// TIA Portal V19 export
FUNCTION_BLOCK "HMI_A04_FB"   // FB117, LAD
TITLE = HMI Managment
AUTHOR : Piemme
FAMILY : System
// stored: MemoryReserve 100, SetENOAutomatically false
   VAR_OUTPUT
      MB4_LpJog : Bool;
   END_VAR
   VAR
      MB4_Decoder { ExternalAccessible := 'False'; ExternalVisible := 'False'; ExternalWritable := 'False'} : "ButtonsHMIDecoder";
   END_VAR
   VAR CONSTANT
      "3002_TRASPORTO" : Int := 3002;
      "3011_FERMI_P1" : Int := 3011;
      "3012_FERMI_P1_SFALSATORE" : Int := 3012;
      "3021_FERMI_P2" : Int := 3021;
      "3022_FERMI_P2_SOLLEVATORE" : Int := 3022;
      "3031_FERMI_P3" : Int := 3031;
      "3032_SOLLEVA_RIBALTA" : Int := 3032;
      "3033_ROT_RIBALTA" : Int := 3033;
      "3041_FERMI_P4" : Int := 3041;
      "3042_SPINTORE_LAT_VRT_P5" : Int := 3042;
      "3043_SPINTORE_LAT_ORZ_P5" : Int := 3043;
      "3044_SOLLEVATORI_P5" : Int := 3044;
      "3045_SPINTORE_LAT_OP" : Int := 3045;
      "3051_RIBALTATORE_OP-POS0" : Int := 3051;
      "3052_RIBALTATORE_OP-POS1" : Int := 3052;
      "3053_RIBALTATORE_OP-POS2" : Int := 3053;
      "3054_RIBALTATORE_OP-POS3" : Int := 3054;
      "4001_HU_CYTROPACK" : Int := 4001;
      "4011_SPINTORE_OP" : Int := 4011;
      "4012_SPINTORE_AX" : Int := 4012;
      "4013_SPINTORE_VRT" : Int := 4013;
      "4014_SPINTORE_ORZ" : Int := 4014;
      "4021_BORDATRICE_AX" : Int := 4021;
      "4031_RULLIERA_OP" : Int := 4031;
      "4032_RULLIERA_AX" : Int := 4032;
      "4033_BORDATRICE_REG-CASSETTA" : Int := 4033;
      "4034_BORDATRICE_PASS01" : Int := 4034;
      "4035_BORDATRICE_PASS02" : Int := 4035;
      "4036_BORDATRICE_PASS03" : Int := 4036;
      "4037_BORDATRICE_PASS04" : Int := 4037;
      "4038_BORDATRICE_REG-CASSETTA_AX-POS" : Int := 4038;
      "4041_CENTRATORI_OP" : Int := 4041;
      "4042_CENTRATORI_CENTRAGGIO" : Int := 4042;
      "4043_CENTRATORI_SOLLEVAMENTO" : Int := 4043;
      "4051_PAREGGIATORE_CODA_OP" : Int := 4051;
      "4052_PAREGGIATORE_CODA_AX" : Int := 4052;
      "4053_PAREGGIATORE_CODA_BLOCCAGGIO" : Int := 4053;
      "4054_PAREGGIATORE_CODA_BATTUTAVERTICALE" : Int := 4054;
      "4055_PAREGGIATORE_CODA_PAREGGIATORELONGIT" : Int := 4055;
      "4061_PAREGGIATORE_TESTA_OP" : Int := 4061;
      "4062_PAREGGIATORE_TESTA_AX" : Int := 4062;
      "4063_PAREGGIATORE_TESTA_BLOCCAGGIO" : Int := 4063;
      "4064_PAREGGIATORE_TESTA_SOLLEVAMENTO" : Int := 4064;
      "4065_PAREGGIATORE_TESTA_CENTRAGGIO" : Int := 4065;
      "4066_PAREGG_TESTA_AX_POS" : Int := 4066;
      "4067_PAREGG_TESTA_AX_POS" : Int := 4067;
      "4071_MANIPOLATORE_AX" : Int := 4071;
      "4072_MANIPOLATORE_AX-POS" : Int := 4072;
      "4073_MANIPOLATORE_MAGNETE" : Int := 4073;
      "4074_MANIPOLATORE_SOLLEVATORE" : Int := 4074;
      "4080_BORDATRICE_PASS01_LATO-OP" : Int := 4080;
      "4081_BORDATRICE_PASS01_LATO-MOT" : Int := 4081;
      "4082_BORDATRICE_PASS02_LATO-OP" : Int := 4082;
      "4083_BORDATRICE_PASS02_LATO-MOT" : Int := 4083;
      "4084_BORDATRICE_PASS03_LATO-OP" : Int := 4084;
      "4085_BORDATRICE_PASS03_LATO-MOT" : Int := 4085;
      "4086_BORDATRICE_PASS04_LATO-OP" : Int := 4086;
      "4087_BORDATRICE_PASS04_LATO-MOT" : Int := 4087;
      "4088_BORDATRICE_PASS01-COMBO_AX-POS" : Int := 4088;
      "4089_BORDATRICE_PASS02-COMBO_AX-POS" : Int := 4089;
      "4090_BORDATRICE_PASS03-COMBO_AX-POS" : Int := 4090;
      "4091_BORDATRICE_PASS04-COMBO_AX-POS" : Int := 4091;
      "4092_BORDATRICE_PASS01-LATO-OP_AX-POS" : Int := 4092;
      "4093_BORDATRICE_PASS01-LATO-MOT_AX-POS" : Int := 4093;
      "4094_BORDATRICE_PASS02-LATO-OP_AX-POS" : Int := 4094;
      "4095_BORDATRICE_PASS02-LATO-MOT_AX-POS" : Int := 4095;
      "4096_BORDATRICE_PASS03-LATO-OP_AX-POS" : Int := 4096;
      "4097_BORDATRICE_PASS03-LATO-MOT_AX-POS" : Int := 4097;
      "4098_BORDATRICE_PASS04-LATO-OP_AX-POS" : Int := 4098;
      "4099_BORDATRICE_PASS04-LATO-MOT_AX-POS" : Int := 4099;
      "5001_SPALLA_OP_POS" : Int := 5001;
      "5002_SPALLA_TESTA_AX_JOG" : Int := 5002;
      "5003_SPALLA_TESTA_AX_POS" : Int := 5003;
      "5005_SPALLA_CODA_AX" : Int := 5005;
      "5006_SPALLA_CODA_AX_POS" : Int := 5006;
      "5011_SPINTORE_OP" : Int := 5011;
      "5012_SPINTORE_VRT" : Int := 5012;
      "5013_SPINTORE_ORZ" : Int := 5013;
      "5021_TRASLAZIONE_OP_VAI_A_PRELIEVO" : Int := 5021;
      "5022_TRASLAZIONE_OP_PRELIEVO" : Int := 5022;
      "5023_TRASLAZIONE_OP_VAI_A_DEPOSITO" : Int := 5023;
      "5024_TRASLAZIONE_OP_DEPOSITO" : Int := 5024;
      "5025_TRASLAZIONE_AX_JOG" : Int := 5025;
      "5026_TRASLAZIONE_AX_POS" : Int := 5026;
      "5027_TRASLAZIONE_MANIP_SOSTEGNO" : Int := 5027;
      "5028_TRASLAZIONE_MANIP_PAREGGIATORE" : Int := 5028;
      "5029_TRASLAZIONE_SOSTEGNO_VERTICALE" : Int := 5029;
      "5031_SOLLEVAMENTO_OP" : Int := 5031;
      "5032_SOLLEVAMENTO_AX_JOG" : Int := 5032;
      "5033_SOLLEVAMENTO_AX_POS" : Int := 5033;
      "5041_PALETTIANTIRIBALTAMENTO_OP" : Int := 5041;
      "5042_PALETTIANTIRIBALTAMENTO_TESTA_POS0" : Int := 5042;
      "5043_PALETTIANTIRIBALTAMENTO_TESTA_POS1" : Int := 5043;
      "5044_PALETTIANTIRIBALTAMENTO_TESTA_POS2" : Int := 5044;
      "5046_PALETTIANTIRIBALTAMENTO_CODA_POS0" : Int := 5046;
      "5047_PALETTIANTIRIBALTAMENTO_CODA_POS1" : Int := 5047;
      "5048_PALETTIANTIRIBALTAMENTO_CODA_POS2" : Int := 5048;
      "5051_SOSTEGNO_TESTA_AX_JOG" : Int := 5051;
      "5052_SOSTEGNO_TESTA_AX_POS" : Int := 5052;
      "5053_SOSTEGNO_CODA_AX_JOG" : Int := 5053;
      "5054_SOSTEGNO_CODA_AX_POS" : Int := 5054;
      "6001_NAVETTA_OP_VAI_A_PRELIEVO" : Int := 6001;
      "6002_NAVETTA_OP_PRELIEVO" : Int := 6002;
      "6003_NAVETTA_OP_VAI_A_DEPOSITO" : Int := 6003;
      "6004_NAVETTA_OP_DEPOSITO" : Int := 6004;
      "6005_NAVETTA_AX" : Int := 6005;
      "6006_NAVETTA_PALETTI_INTERNI" : Int := 6006;
      "6007_NAVETTA_PALETTI_ESTERNI" : Int := 6007;
      "6008_NAVETTA_AX_POS" : Int := 6008;
   END_VAR
   VAR_TEMP   // added for the SCL form of the ladder/FBD networks
      _w1 : Bool;
   END_VAR
BEGIN

REGION Network 2: <<< MB3 MANUALS OPERATIONS >>>
END_REGION

REGION Network 3 (SCL): Reset Op
   #MB4_Decoder.OpEnabled := FALSE;
   #MB4_Decoder.OpRunning := FALSE;
   #MB4_Decoder.OpDone := FALSE;
END_REGION

REGION Network 4: <<<<<<<<< A0303 STAZIONE 3 >>>>>>>>>>>>>
END_REGION

REGION Network 5: MB3 Code 5001- SPALLE - OP
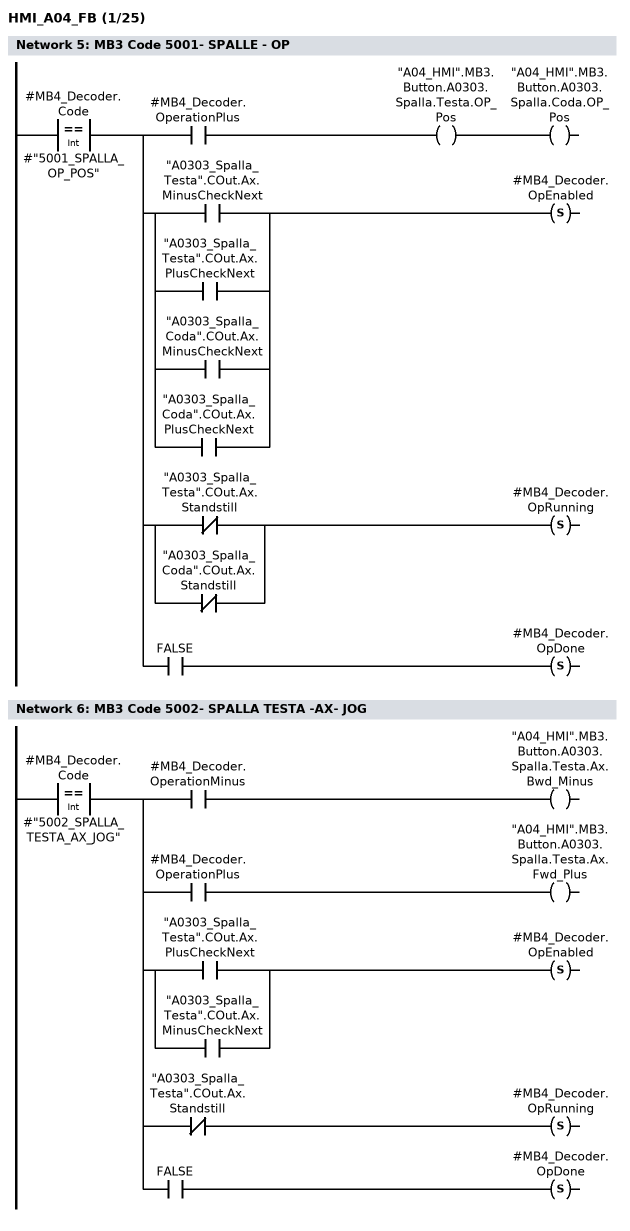
   RUNG wire#powerrail
      { S7_Templates := "SrcType := Int" } EQ_Contact(in1 := #MB4_Decoder.Code, in2 := #"5001_SPALLA_OP_POS")
      wire#w1
      Contact( #MB4_Decoder.OperationPlus )
      Coil( "A04_HMI".MB3.Button.A0303.Spalla.Testa.OP_Pos )
      Coil( "A04_HMI".MB3.Button.A0303.Spalla.Coda.OP_Pos )
   END_RUNG
   RUNG wire#w1
      Contact( "A0303_Spalla_Testa".COut.Ax.MinusCheckNext )
      wire#w2
      S_Coil( #MB4_Decoder.OpEnabled )
   END_RUNG
   RUNG wire#w1
      Contact( "A0303_Spalla_Testa".COut.Ax.PlusCheckNext )
   END_RUNG wire#w2
   RUNG wire#w1
      Contact( "A0303_Spalla_Coda".COut.Ax.MinusCheckNext )
   END_RUNG wire#w2
   RUNG wire#w1
      Contact( "A0303_Spalla_Coda".COut.Ax.PlusCheckNext )
   END_RUNG wire#w2
   RUNG wire#w1
      I_Contact( "A0303_Spalla_Testa".COut.Ax.Standstill )
      wire#w3
      S_Coil( #MB4_Decoder.OpRunning )
   END_RUNG
   RUNG wire#w1
      I_Contact( "A0303_Spalla_Coda".COut.Ax.Standstill )
   END_RUNG wire#w3
   RUNG wire#w1
      Contact( FALSE )
      S_Coil( #MB4_Decoder.OpDone )
   END_RUNG
   // the same network as SCL:
   #_w1 := #MB4_Decoder.Code = #"5001_SPALLA_OP_POS";
   "A04_HMI".MB3.Button.A0303.Spalla.Testa.OP_Pos := #_w1 AND #MB4_Decoder.OperationPlus;
   "A04_HMI".MB3.Button.A0303.Spalla.Coda.OP_Pos := "A04_HMI".MB3.Button.A0303.Spalla.Testa.OP_Pos;
   IF #_w1 AND ("A0303_Spalla_Testa".COut.Ax.MinusCheckNext OR "A0303_Spalla_Testa".COut.Ax.PlusCheckNext OR "A0303_Spalla_Coda".COut.Ax.MinusCheckNext OR "A0303_Spalla_Coda".COut.Ax.PlusCheckNext) THEN
       #MB4_Decoder.OpEnabled := TRUE;
   END_IF;
   IF #_w1 AND (NOT "A0303_Spalla_Testa".COut.Ax.Standstill OR NOT "A0303_Spalla_Coda".COut.Ax.Standstill) THEN
       #MB4_Decoder.OpRunning := TRUE;
   END_IF;
   IF #_w1 AND FALSE THEN #MB4_Decoder.OpDone := TRUE; END_IF;
END_REGION

REGION Network 6: MB3 Code 5002- SPALLA TESTA -AX- JOG
   RUNG wire#powerrail
      { S7_Templates := "SrcType := Int" } EQ_Contact(in1 := #MB4_Decoder.Code, in2 := #"5002_SPALLA_TESTA_AX_JOG")
      wire#w1
      Contact( #MB4_Decoder.OperationMinus )
      Coil( "A04_HMI".MB3.Button.A0303.Spalla.Testa.Ax.Bwd_Minus )
   END_RUNG
   RUNG wire#w1
      Contact( #MB4_Decoder.OperationPlus )
      Coil( "A04_HMI".MB3.Button.A0303.Spalla.Testa.Ax.Fwd_Plus )
   END_RUNG
   RUNG wire#w1
      Contact( "A0303_Spalla_Testa".COut.Ax.PlusCheckNext )
      wire#w2
      S_Coil( #MB4_Decoder.OpEnabled )
   END_RUNG
   RUNG wire#w1
      Contact( "A0303_Spalla_Testa".COut.Ax.MinusCheckNext )
   END_RUNG wire#w2
   RUNG wire#w1
      I_Contact( "A0303_Spalla_Testa".COut.Ax.Standstill )
      S_Coil( #MB4_Decoder.OpRunning )
   END_RUNG
   RUNG wire#w1
      Contact( FALSE )
      S_Coil( #MB4_Decoder.OpDone )
   END_RUNG
   // the same network as SCL:
   #_w1 := #MB4_Decoder.Code = #"5002_SPALLA_TESTA_AX_JOG";
   "A04_HMI".MB3.Button.A0303.Spalla.Testa.Ax.Bwd_Minus := #_w1 AND #MB4_Decoder.OperationMinus;
   "A04_HMI".MB3.Button.A0303.Spalla.Testa.Ax.Fwd_Plus := #_w1 AND #MB4_Decoder.OperationPlus;
   IF #_w1 AND ("A0303_Spalla_Testa".COut.Ax.PlusCheckNext OR "A0303_Spalla_Testa".COut.Ax.MinusCheckNext) THEN
       #MB4_Decoder.OpEnabled := TRUE;
   END_IF;
   IF #_w1 AND NOT "A0303_Spalla_Testa".COut.Ax.Standstill THEN #MB4_Decoder.OpRunning := TRUE; END_IF;
   IF #_w1 AND FALSE THEN #MB4_Decoder.OpDone := TRUE; END_IF;
END_REGION

REGION Network 7: MB3 Code 5003- SPALLA TESTA -AX - POS
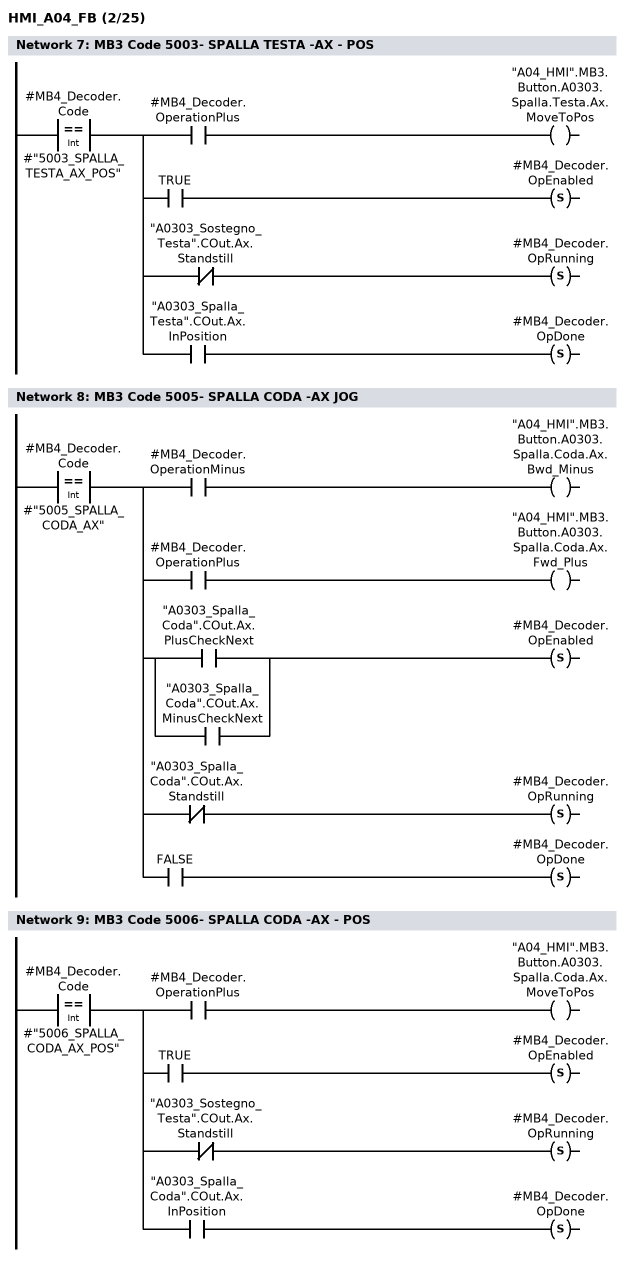
   RUNG wire#powerrail
      { S7_Templates := "SrcType := Int" } EQ_Contact(in1 := #MB4_Decoder.Code, in2 := #"5003_SPALLA_TESTA_AX_POS")
      wire#w1
      Contact( #MB4_Decoder.OperationPlus )
      Coil( "A04_HMI".MB3.Button.A0303.Spalla.Testa.Ax.MoveToPos )
   END_RUNG
   RUNG wire#w1
      Contact( TRUE )
      S_Coil( #MB4_Decoder.OpEnabled )
   END_RUNG
   RUNG wire#w1
      I_Contact( "A0303_Sostegno_Testa".COut.Ax.Standstill )
      S_Coil( #MB4_Decoder.OpRunning )
   END_RUNG
   RUNG wire#w1
      Contact( "A0303_Spalla_Testa".COut.Ax.InPosition )
      S_Coil( #MB4_Decoder.OpDone )
   END_RUNG
   // the same network as SCL:
   #_w1 := #MB4_Decoder.Code = #"5003_SPALLA_TESTA_AX_POS";
   "A04_HMI".MB3.Button.A0303.Spalla.Testa.Ax.MoveToPos := #_w1 AND #MB4_Decoder.OperationPlus;
   IF #_w1 AND TRUE THEN #MB4_Decoder.OpEnabled := TRUE; END_IF;
   IF #_w1 AND NOT "A0303_Sostegno_Testa".COut.Ax.Standstill THEN #MB4_Decoder.OpRunning := TRUE; END_IF;
   IF #_w1 AND "A0303_Spalla_Testa".COut.Ax.InPosition THEN #MB4_Decoder.OpDone := TRUE; END_IF;
END_REGION

REGION Network 8: MB3 Code 5005- SPALLA CODA -AX JOG
   RUNG wire#powerrail
      { S7_Templates := "SrcType := Int" } EQ_Contact(in1 := #MB4_Decoder.Code, in2 := #"5005_SPALLA_CODA_AX")
      wire#w1
      Contact( #MB4_Decoder.OperationMinus )
      Coil( "A04_HMI".MB3.Button.A0303.Spalla.Coda.Ax.Bwd_Minus )
   END_RUNG
   RUNG wire#w1
      Contact( #MB4_Decoder.OperationPlus )
      Coil( "A04_HMI".MB3.Button.A0303.Spalla.Coda.Ax.Fwd_Plus )
   END_RUNG
   RUNG wire#w1
      Contact( "A0303_Spalla_Coda".COut.Ax.PlusCheckNext )
      wire#w2
      S_Coil( #MB4_Decoder.OpEnabled )
   END_RUNG
   RUNG wire#w1
      Contact( "A0303_Spalla_Coda".COut.Ax.MinusCheckNext )
   END_RUNG wire#w2
   RUNG wire#w1
      I_Contact( "A0303_Spalla_Coda".COut.Ax.Standstill )
      S_Coil( #MB4_Decoder.OpRunning )
   END_RUNG
   RUNG wire#w1
      Contact( FALSE )
      S_Coil( #MB4_Decoder.OpDone )
   END_RUNG
   // the same network as SCL:
   #_w1 := #MB4_Decoder.Code = #"5005_SPALLA_CODA_AX";
   "A04_HMI".MB3.Button.A0303.Spalla.Coda.Ax.Bwd_Minus := #_w1 AND #MB4_Decoder.OperationMinus;
   "A04_HMI".MB3.Button.A0303.Spalla.Coda.Ax.Fwd_Plus := #_w1 AND #MB4_Decoder.OperationPlus;
   IF #_w1 AND ("A0303_Spalla_Coda".COut.Ax.PlusCheckNext OR "A0303_Spalla_Coda".COut.Ax.MinusCheckNext) THEN
       #MB4_Decoder.OpEnabled := TRUE;
   END_IF;
   IF #_w1 AND NOT "A0303_Spalla_Coda".COut.Ax.Standstill THEN #MB4_Decoder.OpRunning := TRUE; END_IF;
   IF #_w1 AND FALSE THEN #MB4_Decoder.OpDone := TRUE; END_IF;
END_REGION

REGION Network 9: MB3 Code 5006- SPALLA CODA -AX - POS
   RUNG wire#powerrail
      { S7_Templates := "SrcType := Int" } EQ_Contact(in1 := #MB4_Decoder.Code, in2 := #"5006_SPALLA_CODA_AX_POS")
      wire#w1
      Contact( #MB4_Decoder.OperationPlus )
      Coil( "A04_HMI".MB3.Button.A0303.Spalla.Coda.Ax.MoveToPos )
   END_RUNG
   RUNG wire#w1
      Contact( TRUE )
      S_Coil( #MB4_Decoder.OpEnabled )
   END_RUNG
   RUNG wire#w1
      I_Contact( "A0303_Sostegno_Testa".COut.Ax.Standstill )
      S_Coil( #MB4_Decoder.OpRunning )
   END_RUNG
   RUNG wire#w1
      Contact( "A0303_Spalla_Coda".COut.Ax.InPosition )
      S_Coil( #MB4_Decoder.OpDone )
   END_RUNG
   // the same network as SCL:
   #_w1 := #MB4_Decoder.Code = #"5006_SPALLA_CODA_AX_POS";
   "A04_HMI".MB3.Button.A0303.Spalla.Coda.Ax.MoveToPos := #_w1 AND #MB4_Decoder.OperationPlus;
   IF #_w1 AND TRUE THEN #MB4_Decoder.OpEnabled := TRUE; END_IF;
   IF #_w1 AND NOT "A0303_Sostegno_Testa".COut.Ax.Standstill THEN #MB4_Decoder.OpRunning := TRUE; END_IF;
   IF #_w1 AND "A0303_Spalla_Coda".COut.Ax.InPosition THEN #MB4_Decoder.OpDone := TRUE; END_IF;
END_REGION

REGION Network 10: MB3 Code 5011- SPINTORE- OP
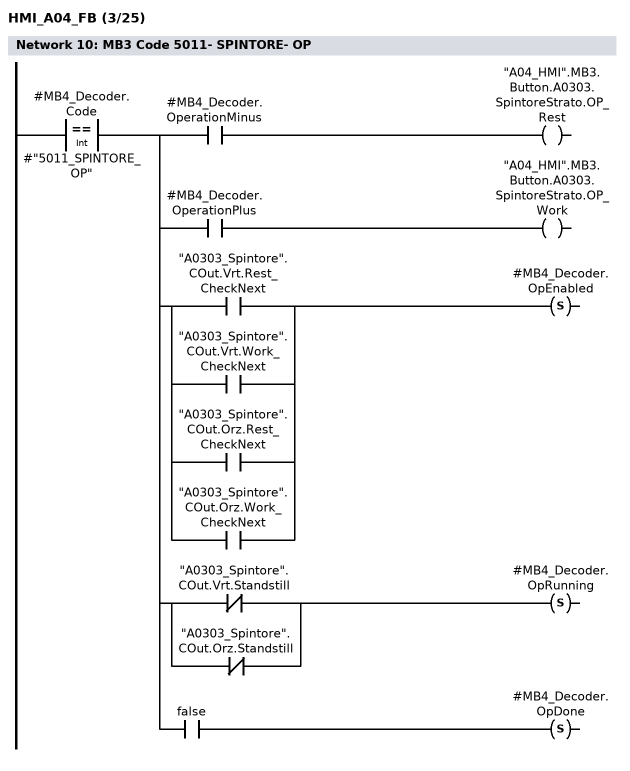
   RUNG wire#powerrail
      { S7_Templates := "SrcType := Int" } EQ_Contact(in1 := #MB4_Decoder.Code, in2 := #"5011_SPINTORE_OP")
      wire#w1
      Contact( #MB4_Decoder.OperationMinus )
      Coil( "A04_HMI".MB3.Button.A0303.SpintoreStrato.OP_Rest )
   END_RUNG
   RUNG wire#w1
      Contact( #MB4_Decoder.OperationPlus )
      Coil( "A04_HMI".MB3.Button.A0303.SpintoreStrato.OP_Work )
   END_RUNG
   RUNG wire#w1
      Contact( "A0303_Spintore".COut.Vrt.Rest_CheckNext )
      wire#w2
      S_Coil( #MB4_Decoder.OpEnabled )
   END_RUNG
   RUNG wire#w1
      Contact( "A0303_Spintore".COut.Vrt.Work_CheckNext )
   END_RUNG wire#w2
   RUNG wire#w1
      Contact( "A0303_Spintore".COut.Orz.Rest_CheckNext )
   END_RUNG wire#w2
   RUNG wire#w1
      Contact( "A0303_Spintore".COut.Orz.Work_CheckNext )
   END_RUNG wire#w2
   RUNG wire#w1
      I_Contact( "A0303_Spintore".COut.Vrt.Standstill )
      wire#w3
      S_Coil( #MB4_Decoder.OpRunning )
   END_RUNG
   RUNG wire#w1
      I_Contact( "A0303_Spintore".COut.Orz.Standstill )
   END_RUNG wire#w3
   RUNG wire#w1
      Contact( false )
      S_Coil( #MB4_Decoder.OpDone )
   END_RUNG
   // the same network as SCL:
   #_w1 := #MB4_Decoder.Code = #"5011_SPINTORE_OP";
   "A04_HMI".MB3.Button.A0303.SpintoreStrato.OP_Rest := #_w1 AND #MB4_Decoder.OperationMinus;
   "A04_HMI".MB3.Button.A0303.SpintoreStrato.OP_Work := #_w1 AND #MB4_Decoder.OperationPlus;
   IF #_w1 AND ("A0303_Spintore".COut.Vrt.Rest_CheckNext OR "A0303_Spintore".COut.Vrt.Work_CheckNext OR "A0303_Spintore".COut.Orz.Rest_CheckNext OR "A0303_Spintore".COut.Orz.Work_CheckNext) THEN
       #MB4_Decoder.OpEnabled := TRUE;
   END_IF;
   IF #_w1 AND (NOT "A0303_Spintore".COut.Vrt.Standstill OR NOT "A0303_Spintore".COut.Orz.Standstill) THEN
       #MB4_Decoder.OpRunning := TRUE;
   END_IF;
   IF #_w1 AND false THEN #MB4_Decoder.OpDone := TRUE; END_IF;
END_REGION

REGION Network 11: MB3 Code 5012 - SPINTORE- VERTICALE
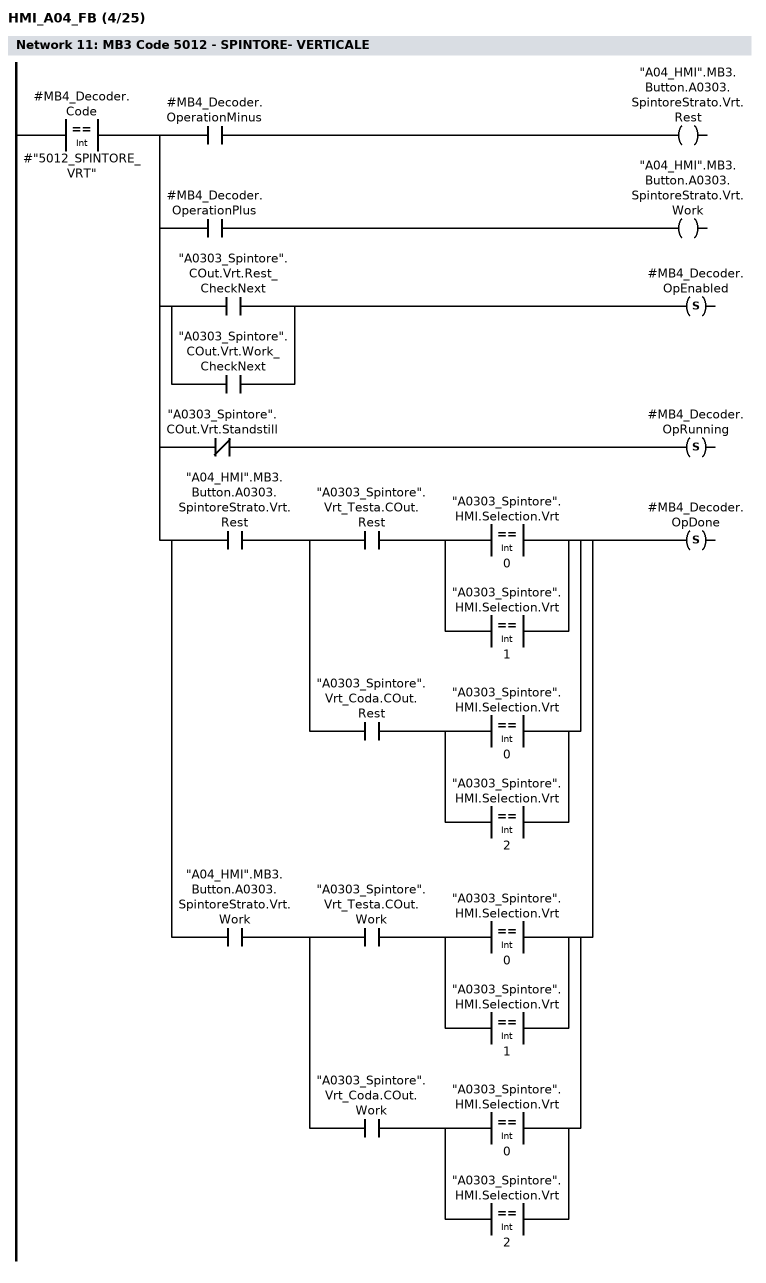
   RUNG wire#powerrail
      { S7_Templates := "SrcType := Int" } EQ_Contact(in1 := #MB4_Decoder.Code, in2 := #"5012_SPINTORE_VRT")
      wire#w1
      Contact( #MB4_Decoder.OperationMinus )
      Coil( "A04_HMI".MB3.Button.A0303.SpintoreStrato.Vrt.Rest )
   END_RUNG
   RUNG wire#w1
      Contact( #MB4_Decoder.OperationPlus )
      Coil( "A04_HMI".MB3.Button.A0303.SpintoreStrato.Vrt.Work )
   END_RUNG
   RUNG wire#w1
      Contact( "A0303_Spintore".COut.Vrt.Rest_CheckNext )
      wire#w2
      S_Coil( #MB4_Decoder.OpEnabled )
   END_RUNG
   RUNG wire#w1
      Contact( "A0303_Spintore".COut.Vrt.Work_CheckNext )
   END_RUNG wire#w2
   RUNG wire#w1
      I_Contact( "A0303_Spintore".COut.Vrt.Standstill )
      S_Coil( #MB4_Decoder.OpRunning )
   END_RUNG
   RUNG wire#w1
      Contact( "A04_HMI".MB3.Button.A0303.SpintoreStrato.Vrt.Rest )
      wire#w3
      Contact( "A0303_Spintore".Vrt_Testa.COut.Rest )
      wire#w4
      { S7_Templates := "SrcType := Int" } EQ_Contact(in1 := "A0303_Spintore".HMI.Selection.Vrt, in2 := 0)
      wire#w5
      S_Coil( #MB4_Decoder.OpDone )
   END_RUNG
   RUNG wire#w4
      { S7_Templates := "SrcType := Int" } EQ_Contact(in1 := "A0303_Spintore".HMI.Selection.Vrt, in2 := 1)
   END_RUNG wire#w5
   RUNG wire#w3
      Contact( "A0303_Spintore".Vrt_Coda.COut.Rest )
      wire#w6
      { S7_Templates := "SrcType := Int" } EQ_Contact(in1 := "A0303_Spintore".HMI.Selection.Vrt, in2 := 0)
   END_RUNG wire#w5
   RUNG wire#w6
      { S7_Templates := "SrcType := Int" } EQ_Contact(in1 := "A0303_Spintore".HMI.Selection.Vrt, in2 := 2)
   END_RUNG wire#w5
   RUNG wire#w1
      Contact( "A04_HMI".MB3.Button.A0303.SpintoreStrato.Vrt.Work )
      wire#w7
      Contact( "A0303_Spintore".Vrt_Testa.COut.Work )
      wire#w8
      { S7_Templates := "SrcType := Int" } EQ_Contact(in1 := "A0303_Spintore".HMI.Selection.Vrt, in2 := 0)
   END_RUNG wire#w5
   RUNG wire#w8
      { S7_Templates := "SrcType := Int" } EQ_Contact(in1 := "A0303_Spintore".HMI.Selection.Vrt, in2 := 1)
   END_RUNG wire#w5
   RUNG wire#w7
      Contact( "A0303_Spintore".Vrt_Coda.COut.Work )
      wire#w9
      { S7_Templates := "SrcType := Int" } EQ_Contact(in1 := "A0303_Spintore".HMI.Selection.Vrt, in2 := 0)
   END_RUNG wire#w5
   RUNG wire#w9
      { S7_Templates := "SrcType := Int" } EQ_Contact(in1 := "A0303_Spintore".HMI.Selection.Vrt, in2 := 2)
   END_RUNG wire#w5
   // the same network as SCL:
   #_w1 := #MB4_Decoder.Code = #"5012_SPINTORE_VRT";
   "A04_HMI".MB3.Button.A0303.SpintoreStrato.Vrt.Rest := #_w1 AND #MB4_Decoder.OperationMinus;
   "A04_HMI".MB3.Button.A0303.SpintoreStrato.Vrt.Work := #_w1 AND #MB4_Decoder.OperationPlus;
   IF #_w1 AND ("A0303_Spintore".COut.Vrt.Rest_CheckNext OR "A0303_Spintore".COut.Vrt.Work_CheckNext) THEN
       #MB4_Decoder.OpEnabled := TRUE;
   END_IF;
   IF #_w1 AND NOT "A0303_Spintore".COut.Vrt.Standstill THEN #MB4_Decoder.OpRunning := TRUE; END_IF;
   IF #_w1 AND (("A04_HMI".MB3.Button.A0303.SpintoreStrato.Vrt.Rest AND (("A0303_Spintore".Vrt_Testa.COut.Rest AND (("A0303_Spintore".HMI.Selection.Vrt = 0) OR ("A0303_Spintore".HMI.Selection.Vrt = 1))) OR ("A0303_Spintore".Vrt_Coda.COut.Rest AND (("A0303_Spintore".HMI.Selection.Vrt = 0) OR ("A0303_Spintore".HMI.Selection.Vrt = 2))))) OR ("A04_HMI".MB3.Button.A0303.SpintoreStrato.Vrt.Work AND (("A0303_Spintore".Vrt_Testa.COut.Work AND (("A0303_Spintore".HMI.Selection.Vrt = 0) OR ("A0303_Spintore".HMI.Selection.Vrt = 1))) OR ("A0303_Spintore".Vrt_Coda.COut.Work AND (("A0303_Spintore".HMI.Selection.Vrt = 0) OR ("A0303_Spintore".HMI.Selection.Vrt = 2)))))) THEN
       #MB4_Decoder.OpDone := TRUE;
   END_IF;
END_REGION

REGION Network 12: MB3 Code 5013 - SPINTORE- ORIZZONTALE
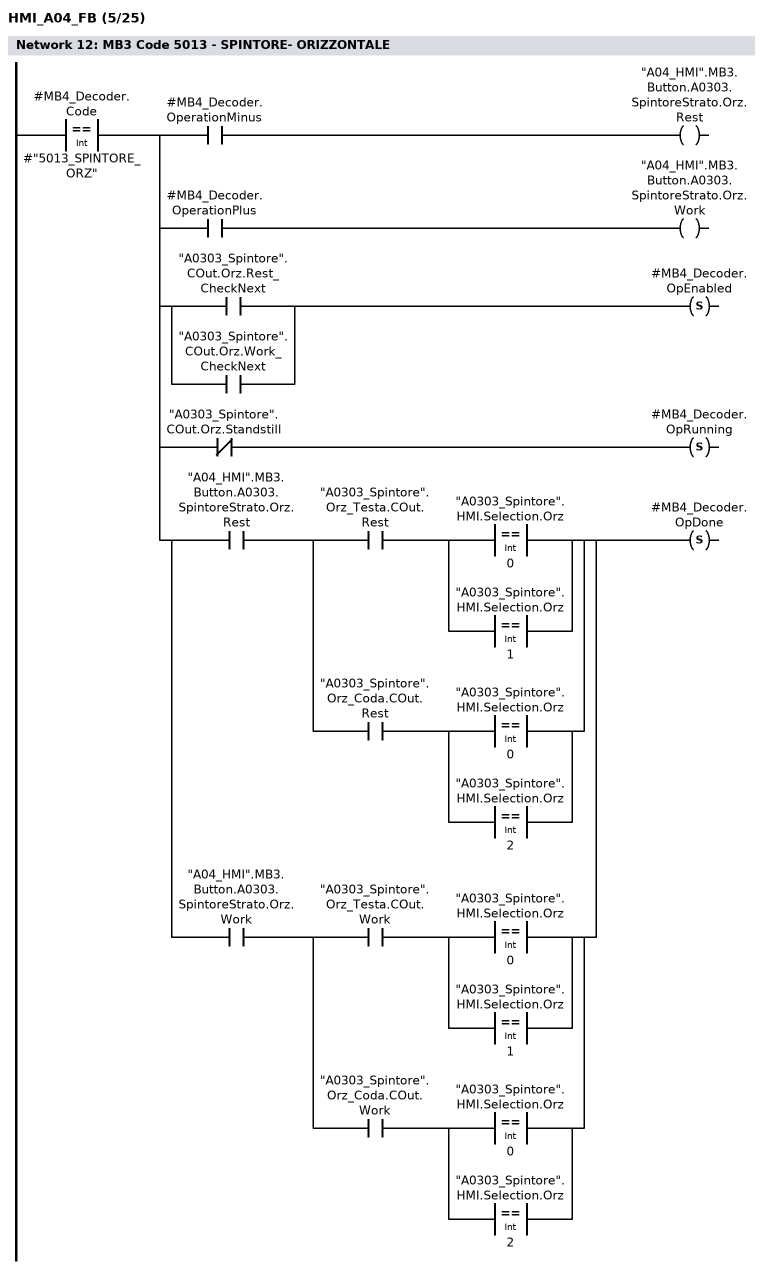
   RUNG wire#powerrail
      { S7_Templates := "SrcType := Int" } EQ_Contact(in1 := #MB4_Decoder.Code, in2 := #"5013_SPINTORE_ORZ")
      wire#w1
      Contact( #MB4_Decoder.OperationMinus )
      Coil( "A04_HMI".MB3.Button.A0303.SpintoreStrato.Orz.Rest )
   END_RUNG
   RUNG wire#w1
      Contact( #MB4_Decoder.OperationPlus )
      Coil( "A04_HMI".MB3.Button.A0303.SpintoreStrato.Orz.Work )
   END_RUNG
   RUNG wire#w1
      Contact( "A0303_Spintore".COut.Orz.Rest_CheckNext )
      wire#w2
      S_Coil( #MB4_Decoder.OpEnabled )
   END_RUNG
   RUNG wire#w1
      Contact( "A0303_Spintore".COut.Orz.Work_CheckNext )
   END_RUNG wire#w2
   RUNG wire#w1
      I_Contact( "A0303_Spintore".COut.Orz.Standstill )
      S_Coil( #MB4_Decoder.OpRunning )
   END_RUNG
   RUNG wire#w1
      Contact( "A04_HMI".MB3.Button.A0303.SpintoreStrato.Orz.Rest )
      wire#w3
      Contact( "A0303_Spintore".Orz_Testa.COut.Rest )
      wire#w4
      { S7_Templates := "SrcType := Int" } EQ_Contact(in1 := "A0303_Spintore".HMI.Selection.Orz, in2 := 0)
      wire#w5
      S_Coil( #MB4_Decoder.OpDone )
   END_RUNG
   RUNG wire#w4
      { S7_Templates := "SrcType := Int" } EQ_Contact(in1 := "A0303_Spintore".HMI.Selection.Orz, in2 := 1)
   END_RUNG wire#w5
   RUNG wire#w3
      Contact( "A0303_Spintore".Orz_Coda.COut.Rest )
      wire#w6
      { S7_Templates := "SrcType := Int" } EQ_Contact(in1 := "A0303_Spintore".HMI.Selection.Orz, in2 := 0)
   END_RUNG wire#w5
   RUNG wire#w6
      { S7_Templates := "SrcType := Int" } EQ_Contact(in1 := "A0303_Spintore".HMI.Selection.Orz, in2 := 2)
   END_RUNG wire#w5
   RUNG wire#w1
      Contact( "A04_HMI".MB3.Button.A0303.SpintoreStrato.Orz.Work )
      wire#w7
      Contact( "A0303_Spintore".Orz_Testa.COut.Work )
      wire#w8
      { S7_Templates := "SrcType := Int" } EQ_Contact(in1 := "A0303_Spintore".HMI.Selection.Orz, in2 := 0)
   END_RUNG wire#w5
   RUNG wire#w8
      { S7_Templates := "SrcType := Int" } EQ_Contact(in1 := "A0303_Spintore".HMI.Selection.Orz, in2 := 1)
   END_RUNG wire#w5
   RUNG wire#w7
      Contact( "A0303_Spintore".Orz_Coda.COut.Work )
      wire#w9
      { S7_Templates := "SrcType := Int" } EQ_Contact(in1 := "A0303_Spintore".HMI.Selection.Orz, in2 := 0)
   END_RUNG wire#w5
   RUNG wire#w9
      { S7_Templates := "SrcType := Int" } EQ_Contact(in1 := "A0303_Spintore".HMI.Selection.Orz, in2 := 2)
   END_RUNG wire#w5
   // the same network as SCL:
   #_w1 := #MB4_Decoder.Code = #"5013_SPINTORE_ORZ";
   "A04_HMI".MB3.Button.A0303.SpintoreStrato.Orz.Rest := #_w1 AND #MB4_Decoder.OperationMinus;
   "A04_HMI".MB3.Button.A0303.SpintoreStrato.Orz.Work := #_w1 AND #MB4_Decoder.OperationPlus;
   IF #_w1 AND ("A0303_Spintore".COut.Orz.Rest_CheckNext OR "A0303_Spintore".COut.Orz.Work_CheckNext) THEN
       #MB4_Decoder.OpEnabled := TRUE;
   END_IF;
   IF #_w1 AND NOT "A0303_Spintore".COut.Orz.Standstill THEN #MB4_Decoder.OpRunning := TRUE; END_IF;
   IF #_w1 AND (("A04_HMI".MB3.Button.A0303.SpintoreStrato.Orz.Rest AND (("A0303_Spintore".Orz_Testa.COut.Rest AND (("A0303_Spintore".HMI.Selection.Orz = 0) OR ("A0303_Spintore".HMI.Selection.Orz = 1))) OR ("A0303_Spintore".Orz_Coda.COut.Rest AND (("A0303_Spintore".HMI.Selection.Orz = 0) OR ("A0303_Spintore".HMI.Selection.Orz = 2))))) OR ("A04_HMI".MB3.Button.A0303.SpintoreStrato.Orz.Work AND (("A0303_Spintore".Orz_Testa.COut.Work AND (("A0303_Spintore".HMI.Selection.Orz = 0) OR ("A0303_Spintore".HMI.Selection.Orz = 1))) OR ("A0303_Spintore".Orz_Coda.COut.Work AND (("A0303_Spintore".HMI.Selection.Orz = 0) OR ("A0303_Spintore".HMI.Selection.Orz = 2)))))) THEN
       #MB4_Decoder.OpDone := TRUE;
   END_IF;
END_REGION

REGION Network 13: MB3 Code 5021- TRASLAZIONE - OP VAI A PRELIEVO
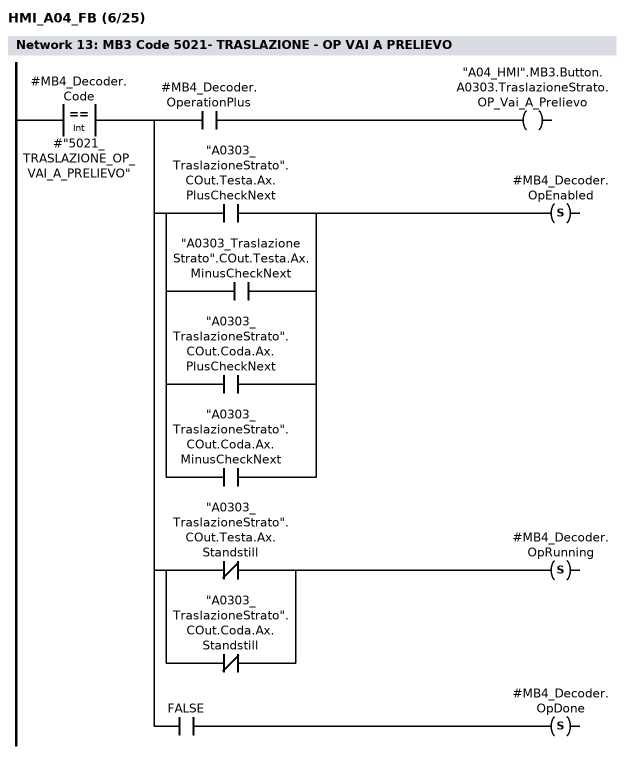
   RUNG wire#powerrail
      { S7_Templates := "SrcType := Int" } EQ_Contact(in1 := #MB4_Decoder.Code, in2 := #"5021_TRASLAZIONE_OP_VAI_A_PRELIEVO")
      wire#w1
      Contact( #MB4_Decoder.OperationPlus )
      Coil( "A04_HMI".MB3.Button.A0303.TraslazioneStrato.OP_Vai_A_Prelievo )
   END_RUNG
   RUNG wire#w1
      Contact( "A0303_TraslazioneStrato".COut.Testa.Ax.PlusCheckNext )
      wire#w2
      S_Coil( #MB4_Decoder.OpEnabled )
   END_RUNG
   RUNG wire#w1
      Contact( "A0303_TraslazioneStrato".COut.Testa.Ax.MinusCheckNext )
   END_RUNG wire#w2
   RUNG wire#w1
      Contact( "A0303_TraslazioneStrato".COut.Coda.Ax.PlusCheckNext )
   END_RUNG wire#w2
   RUNG wire#w1
      Contact( "A0303_TraslazioneStrato".COut.Coda.Ax.MinusCheckNext )
   END_RUNG wire#w2
   RUNG wire#w1
      I_Contact( "A0303_TraslazioneStrato".COut.Testa.Ax.Standstill )
      wire#w3
      S_Coil( #MB4_Decoder.OpRunning )
   END_RUNG
   RUNG wire#w1
      I_Contact( "A0303_TraslazioneStrato".COut.Coda.Ax.Standstill )
   END_RUNG wire#w3
   RUNG wire#w1
      Contact( FALSE )
      S_Coil( #MB4_Decoder.OpDone )
   END_RUNG
   // the same network as SCL:
   #_w1 := #MB4_Decoder.Code = #"5021_TRASLAZIONE_OP_VAI_A_PRELIEVO";
   "A04_HMI".MB3.Button.A0303.TraslazioneStrato.OP_Vai_A_Prelievo := #_w1 AND #MB4_Decoder.OperationPlus;
   IF #_w1 AND ("A0303_TraslazioneStrato".COut.Testa.Ax.PlusCheckNext OR "A0303_TraslazioneStrato".COut.Testa.Ax.MinusCheckNext OR "A0303_TraslazioneStrato".COut.Coda.Ax.PlusCheckNext OR "A0303_TraslazioneStrato".COut.Coda.Ax.MinusCheckNext) THEN
       #MB4_Decoder.OpEnabled := TRUE;
   END_IF;
   IF #_w1 AND (NOT "A0303_TraslazioneStrato".COut.Testa.Ax.Standstill OR NOT "A0303_TraslazioneStrato".COut.Coda.Ax.Standstill) THEN
       #MB4_Decoder.OpRunning := TRUE;
   END_IF;
   IF #_w1 AND FALSE THEN #MB4_Decoder.OpDone := TRUE; END_IF;
END_REGION

REGION Network 14: MB3 Code 5022- TRASLAZIONE - OP PRELIEVO
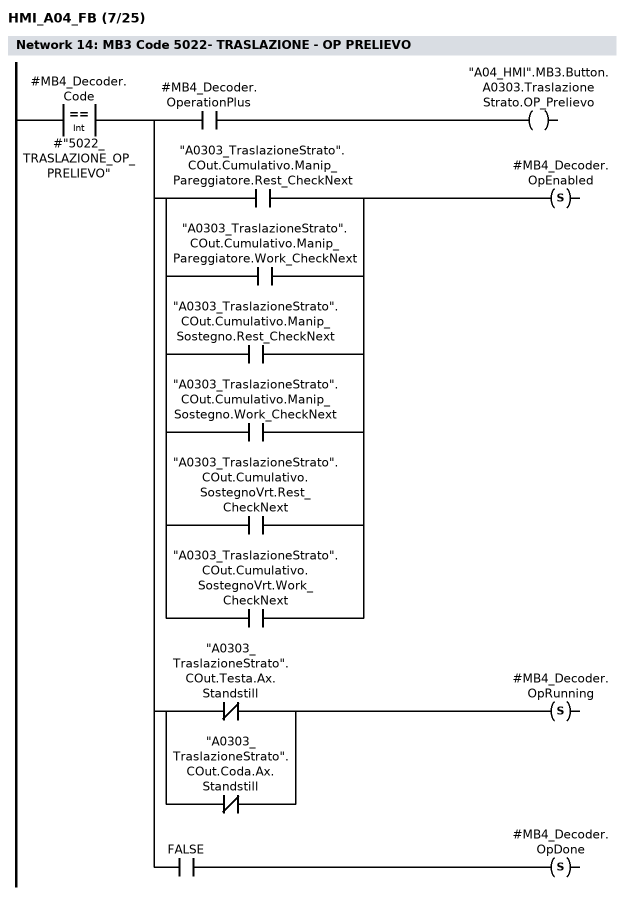
   RUNG wire#powerrail
      { S7_Templates := "SrcType := Int" } EQ_Contact(in1 := #MB4_Decoder.Code, in2 := #"5022_TRASLAZIONE_OP_PRELIEVO")
      wire#w1
      Contact( #MB4_Decoder.OperationPlus )
      Coil( "A04_HMI".MB3.Button.A0303.TraslazioneStrato.OP_Prelievo )
   END_RUNG
   RUNG wire#w1
      Contact( "A0303_TraslazioneStrato".COut.Cumulativo.Manip_Pareggiatore.Rest_CheckNext )
      wire#w2
      S_Coil( #MB4_Decoder.OpEnabled )
   END_RUNG
   RUNG wire#w1
      Contact( "A0303_TraslazioneStrato".COut.Cumulativo.Manip_Pareggiatore.Work_CheckNext )
   END_RUNG wire#w2
   RUNG wire#w1
      Contact( "A0303_TraslazioneStrato".COut.Cumulativo.Manip_Sostegno.Rest_CheckNext )
   END_RUNG wire#w2
   RUNG wire#w1
      Contact( "A0303_TraslazioneStrato".COut.Cumulativo.Manip_Sostegno.Work_CheckNext )
   END_RUNG wire#w2
   RUNG wire#w1
      Contact( "A0303_TraslazioneStrato".COut.Cumulativo.SostegnoVrt.Rest_CheckNext )
   END_RUNG wire#w2
   RUNG wire#w1
      Contact( "A0303_TraslazioneStrato".COut.Cumulativo.SostegnoVrt.Work_CheckNext )
   END_RUNG wire#w2
   RUNG wire#w1
      I_Contact( "A0303_TraslazioneStrato".COut.Testa.Ax.Standstill )
      wire#w3
      S_Coil( #MB4_Decoder.OpRunning )
   END_RUNG
   RUNG wire#w1
      I_Contact( "A0303_TraslazioneStrato".COut.Coda.Ax.Standstill )
   END_RUNG wire#w3
   RUNG wire#w1
      Contact( FALSE )
      S_Coil( #MB4_Decoder.OpDone )
   END_RUNG
   // the same network as SCL:
   #_w1 := #MB4_Decoder.Code = #"5022_TRASLAZIONE_OP_PRELIEVO";
   "A04_HMI".MB3.Button.A0303.TraslazioneStrato.OP_Prelievo := #_w1 AND #MB4_Decoder.OperationPlus;
   IF #_w1 AND ("A0303_TraslazioneStrato".COut.Cumulativo.Manip_Pareggiatore.Rest_CheckNext OR "A0303_TraslazioneStrato".COut.Cumulativo.Manip_Pareggiatore.Work_CheckNext OR "A0303_TraslazioneStrato".COut.Cumulativo.Manip_Sostegno.Rest_CheckNext OR "A0303_TraslazioneStrato".COut.Cumulativo.Manip_Sostegno.Work_CheckNext OR "A0303_TraslazioneStrato".COut.Cumulativo.SostegnoVrt.Rest_CheckNext OR "A0303_TraslazioneStrato".COut.Cumulativo.SostegnoVrt.Work_CheckNext) THEN
       #MB4_Decoder.OpEnabled := TRUE;
   END_IF;
   IF #_w1 AND (NOT "A0303_TraslazioneStrato".COut.Testa.Ax.Standstill OR NOT "A0303_TraslazioneStrato".COut.Coda.Ax.Standstill) THEN
       #MB4_Decoder.OpRunning := TRUE;
   END_IF;
   IF #_w1 AND FALSE THEN #MB4_Decoder.OpDone := TRUE; END_IF;
END_REGION

REGION Network 15: MB3 Code 5023- TRASLAZIONE - OP VAI A DEPOSITO
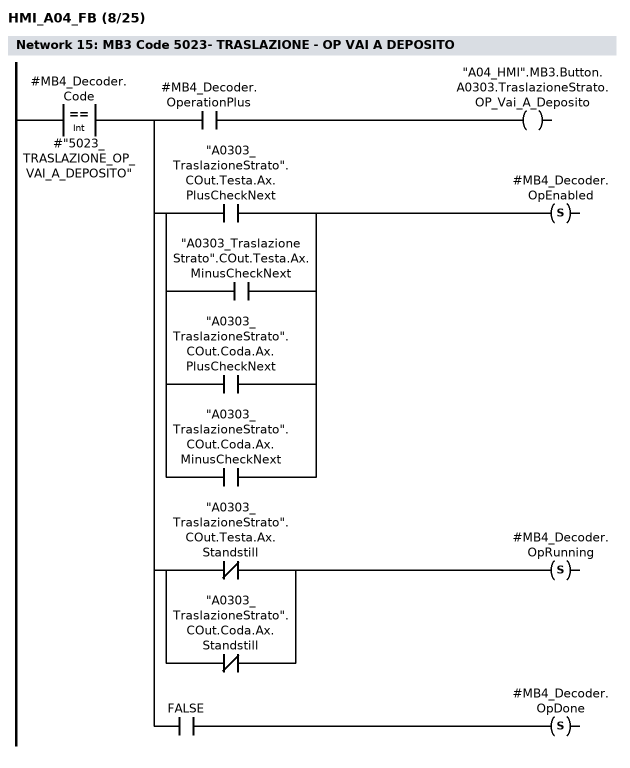
   RUNG wire#powerrail
      { S7_Templates := "SrcType := Int" } EQ_Contact(in1 := #MB4_Decoder.Code, in2 := #"5023_TRASLAZIONE_OP_VAI_A_DEPOSITO")
      wire#w1
      Contact( #MB4_Decoder.OperationPlus )
      Coil( "A04_HMI".MB3.Button.A0303.TraslazioneStrato.OP_Vai_A_Deposito )
   END_RUNG
   RUNG wire#w1
      Contact( "A0303_TraslazioneStrato".COut.Testa.Ax.PlusCheckNext )
      wire#w2
      S_Coil( #MB4_Decoder.OpEnabled )
   END_RUNG
   RUNG wire#w1
      Contact( "A0303_TraslazioneStrato".COut.Testa.Ax.MinusCheckNext )
   END_RUNG wire#w2
   RUNG wire#w1
      Contact( "A0303_TraslazioneStrato".COut.Coda.Ax.PlusCheckNext )
   END_RUNG wire#w2
   RUNG wire#w1
      Contact( "A0303_TraslazioneStrato".COut.Coda.Ax.MinusCheckNext )
   END_RUNG wire#w2
   RUNG wire#w1
      I_Contact( "A0303_TraslazioneStrato".COut.Testa.Ax.Standstill )
      wire#w3
      S_Coil( #MB4_Decoder.OpRunning )
   END_RUNG
   RUNG wire#w1
      I_Contact( "A0303_TraslazioneStrato".COut.Coda.Ax.Standstill )
   END_RUNG wire#w3
   RUNG wire#w1
      Contact( FALSE )
      S_Coil( #MB4_Decoder.OpDone )
   END_RUNG
   // the same network as SCL:
   #_w1 := #MB4_Decoder.Code = #"5023_TRASLAZIONE_OP_VAI_A_DEPOSITO";
   "A04_HMI".MB3.Button.A0303.TraslazioneStrato.OP_Vai_A_Deposito := #_w1 AND #MB4_Decoder.OperationPlus;
   IF #_w1 AND ("A0303_TraslazioneStrato".COut.Testa.Ax.PlusCheckNext OR "A0303_TraslazioneStrato".COut.Testa.Ax.MinusCheckNext OR "A0303_TraslazioneStrato".COut.Coda.Ax.PlusCheckNext OR "A0303_TraslazioneStrato".COut.Coda.Ax.MinusCheckNext) THEN
       #MB4_Decoder.OpEnabled := TRUE;
   END_IF;
   IF #_w1 AND (NOT "A0303_TraslazioneStrato".COut.Testa.Ax.Standstill OR NOT "A0303_TraslazioneStrato".COut.Coda.Ax.Standstill) THEN
       #MB4_Decoder.OpRunning := TRUE;
   END_IF;
   IF #_w1 AND FALSE THEN #MB4_Decoder.OpDone := TRUE; END_IF;
END_REGION

REGION Network 16: MB3 Code 5024- TRASLAZIONE - OP DEPOSITO
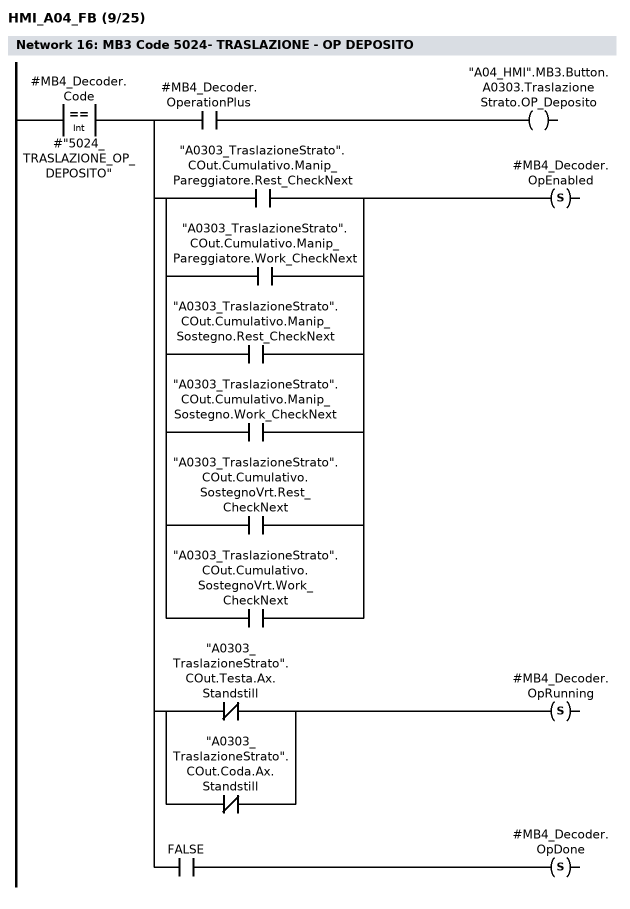
   RUNG wire#powerrail
      { S7_Templates := "SrcType := Int" } EQ_Contact(in1 := #MB4_Decoder.Code, in2 := #"5024_TRASLAZIONE_OP_DEPOSITO")
      wire#w1
      Contact( #MB4_Decoder.OperationPlus )
      Coil( "A04_HMI".MB3.Button.A0303.TraslazioneStrato.OP_Deposito )
   END_RUNG
   RUNG wire#w1
      Contact( "A0303_TraslazioneStrato".COut.Cumulativo.Manip_Pareggiatore.Rest_CheckNext )
      wire#w2
      S_Coil( #MB4_Decoder.OpEnabled )
   END_RUNG
   RUNG wire#w1
      Contact( "A0303_TraslazioneStrato".COut.Cumulativo.Manip_Pareggiatore.Work_CheckNext )
   END_RUNG wire#w2
   RUNG wire#w1
      Contact( "A0303_TraslazioneStrato".COut.Cumulativo.Manip_Sostegno.Rest_CheckNext )
   END_RUNG wire#w2
   RUNG wire#w1
      Contact( "A0303_TraslazioneStrato".COut.Cumulativo.Manip_Sostegno.Work_CheckNext )
   END_RUNG wire#w2
   RUNG wire#w1
      Contact( "A0303_TraslazioneStrato".COut.Cumulativo.SostegnoVrt.Rest_CheckNext )
   END_RUNG wire#w2
   RUNG wire#w1
      Contact( "A0303_TraslazioneStrato".COut.Cumulativo.SostegnoVrt.Work_CheckNext )
   END_RUNG wire#w2
   RUNG wire#w1
      I_Contact( "A0303_TraslazioneStrato".COut.Testa.Ax.Standstill )
      wire#w3
      S_Coil( #MB4_Decoder.OpRunning )
   END_RUNG
   RUNG wire#w1
      I_Contact( "A0303_TraslazioneStrato".COut.Coda.Ax.Standstill )
   END_RUNG wire#w3
   RUNG wire#w1
      Contact( FALSE )
      S_Coil( #MB4_Decoder.OpDone )
   END_RUNG
   // the same network as SCL:
   #_w1 := #MB4_Decoder.Code = #"5024_TRASLAZIONE_OP_DEPOSITO";
   "A04_HMI".MB3.Button.A0303.TraslazioneStrato.OP_Deposito := #_w1 AND #MB4_Decoder.OperationPlus;
   IF #_w1 AND ("A0303_TraslazioneStrato".COut.Cumulativo.Manip_Pareggiatore.Rest_CheckNext OR "A0303_TraslazioneStrato".COut.Cumulativo.Manip_Pareggiatore.Work_CheckNext OR "A0303_TraslazioneStrato".COut.Cumulativo.Manip_Sostegno.Rest_CheckNext OR "A0303_TraslazioneStrato".COut.Cumulativo.Manip_Sostegno.Work_CheckNext OR "A0303_TraslazioneStrato".COut.Cumulativo.SostegnoVrt.Rest_CheckNext OR "A0303_TraslazioneStrato".COut.Cumulativo.SostegnoVrt.Work_CheckNext) THEN
       #MB4_Decoder.OpEnabled := TRUE;
   END_IF;
   IF #_w1 AND (NOT "A0303_TraslazioneStrato".COut.Testa.Ax.Standstill OR NOT "A0303_TraslazioneStrato".COut.Coda.Ax.Standstill) THEN
       #MB4_Decoder.OpRunning := TRUE;
   END_IF;
   IF #_w1 AND FALSE THEN #MB4_Decoder.OpDone := TRUE; END_IF;
END_REGION

REGION Network 17: MB3 Code 5025- TRASLAZIONE -AX - JOG
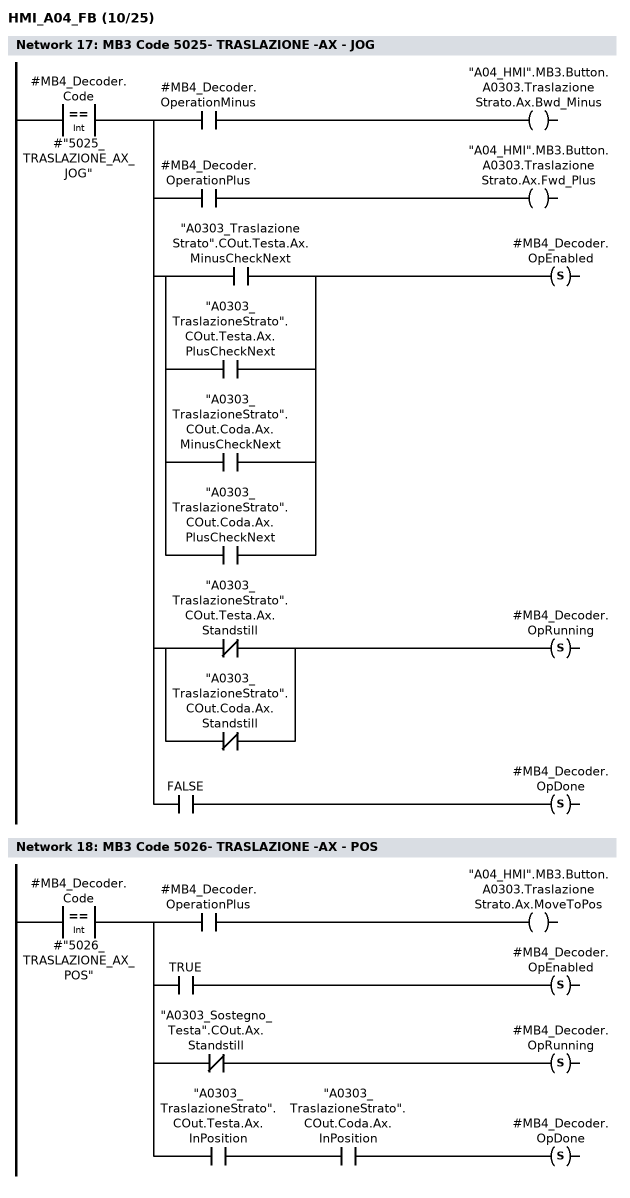
   RUNG wire#powerrail
      { S7_Templates := "SrcType := Int" } EQ_Contact(in1 := #MB4_Decoder.Code, in2 := #"5025_TRASLAZIONE_AX_JOG")
      wire#w1
      Contact( #MB4_Decoder.OperationMinus )
      Coil( "A04_HMI".MB3.Button.A0303.TraslazioneStrato.Ax.Bwd_Minus )
   END_RUNG
   RUNG wire#w1
      Contact( #MB4_Decoder.OperationPlus )
      Coil( "A04_HMI".MB3.Button.A0303.TraslazioneStrato.Ax.Fwd_Plus )
   END_RUNG
   RUNG wire#w1
      Contact( "A0303_TraslazioneStrato".COut.Testa.Ax.MinusCheckNext )
      wire#w2
      S_Coil( #MB4_Decoder.OpEnabled )
   END_RUNG
   RUNG wire#w1
      Contact( "A0303_TraslazioneStrato".COut.Testa.Ax.PlusCheckNext )
   END_RUNG wire#w2
   RUNG wire#w1
      Contact( "A0303_TraslazioneStrato".COut.Coda.Ax.MinusCheckNext )
   END_RUNG wire#w2
   RUNG wire#w1
      Contact( "A0303_TraslazioneStrato".COut.Coda.Ax.PlusCheckNext )
   END_RUNG wire#w2
   RUNG wire#w1
      I_Contact( "A0303_TraslazioneStrato".COut.Testa.Ax.Standstill )
      wire#w3
      S_Coil( #MB4_Decoder.OpRunning )
   END_RUNG
   RUNG wire#w1
      I_Contact( "A0303_TraslazioneStrato".COut.Coda.Ax.Standstill )
   END_RUNG wire#w3
   RUNG wire#w1
      Contact( FALSE )
      S_Coil( #MB4_Decoder.OpDone )
   END_RUNG
   // the same network as SCL:
   #_w1 := #MB4_Decoder.Code = #"5025_TRASLAZIONE_AX_JOG";
   "A04_HMI".MB3.Button.A0303.TraslazioneStrato.Ax.Bwd_Minus := #_w1 AND #MB4_Decoder.OperationMinus;
   "A04_HMI".MB3.Button.A0303.TraslazioneStrato.Ax.Fwd_Plus := #_w1 AND #MB4_Decoder.OperationPlus;
   IF #_w1 AND ("A0303_TraslazioneStrato".COut.Testa.Ax.MinusCheckNext OR "A0303_TraslazioneStrato".COut.Testa.Ax.PlusCheckNext OR "A0303_TraslazioneStrato".COut.Coda.Ax.MinusCheckNext OR "A0303_TraslazioneStrato".COut.Coda.Ax.PlusCheckNext) THEN
       #MB4_Decoder.OpEnabled := TRUE;
   END_IF;
   IF #_w1 AND (NOT "A0303_TraslazioneStrato".COut.Testa.Ax.Standstill OR NOT "A0303_TraslazioneStrato".COut.Coda.Ax.Standstill) THEN
       #MB4_Decoder.OpRunning := TRUE;
   END_IF;
   IF #_w1 AND FALSE THEN #MB4_Decoder.OpDone := TRUE; END_IF;
END_REGION

REGION Network 18: MB3 Code 5026- TRASLAZIONE -AX - POS
   RUNG wire#powerrail
      { S7_Templates := "SrcType := Int" } EQ_Contact(in1 := #MB4_Decoder.Code, in2 := #"5026_TRASLAZIONE_AX_POS")
      wire#w1
      Contact( #MB4_Decoder.OperationPlus )
      Coil( "A04_HMI".MB3.Button.A0303.TraslazioneStrato.Ax.MoveToPos )
   END_RUNG
   RUNG wire#w1
      Contact( TRUE )
      S_Coil( #MB4_Decoder.OpEnabled )
   END_RUNG
   RUNG wire#w1
      I_Contact( "A0303_Sostegno_Testa".COut.Ax.Standstill )
      S_Coil( #MB4_Decoder.OpRunning )
   END_RUNG
   RUNG wire#w1
      Contact( "A0303_TraslazioneStrato".COut.Testa.Ax.InPosition )
      Contact( "A0303_TraslazioneStrato".COut.Coda.Ax.InPosition )
      S_Coil( #MB4_Decoder.OpDone )
   END_RUNG
   // the same network as SCL:
   #_w1 := #MB4_Decoder.Code = #"5026_TRASLAZIONE_AX_POS";
   "A04_HMI".MB3.Button.A0303.TraslazioneStrato.Ax.MoveToPos := #_w1 AND #MB4_Decoder.OperationPlus;
   IF #_w1 AND TRUE THEN #MB4_Decoder.OpEnabled := TRUE; END_IF;
   IF #_w1 AND NOT "A0303_Sostegno_Testa".COut.Ax.Standstill THEN #MB4_Decoder.OpRunning := TRUE; END_IF;
   IF #_w1 AND "A0303_TraslazioneStrato".COut.Testa.Ax.InPosition AND "A0303_TraslazioneStrato".COut.Coda.Ax.InPosition THEN
       #MB4_Decoder.OpDone := TRUE;
   END_IF;
END_REGION

REGION Network 19: MB3 Code 5027 - TRASLAZIONE- MANIP SOSTEGNO L
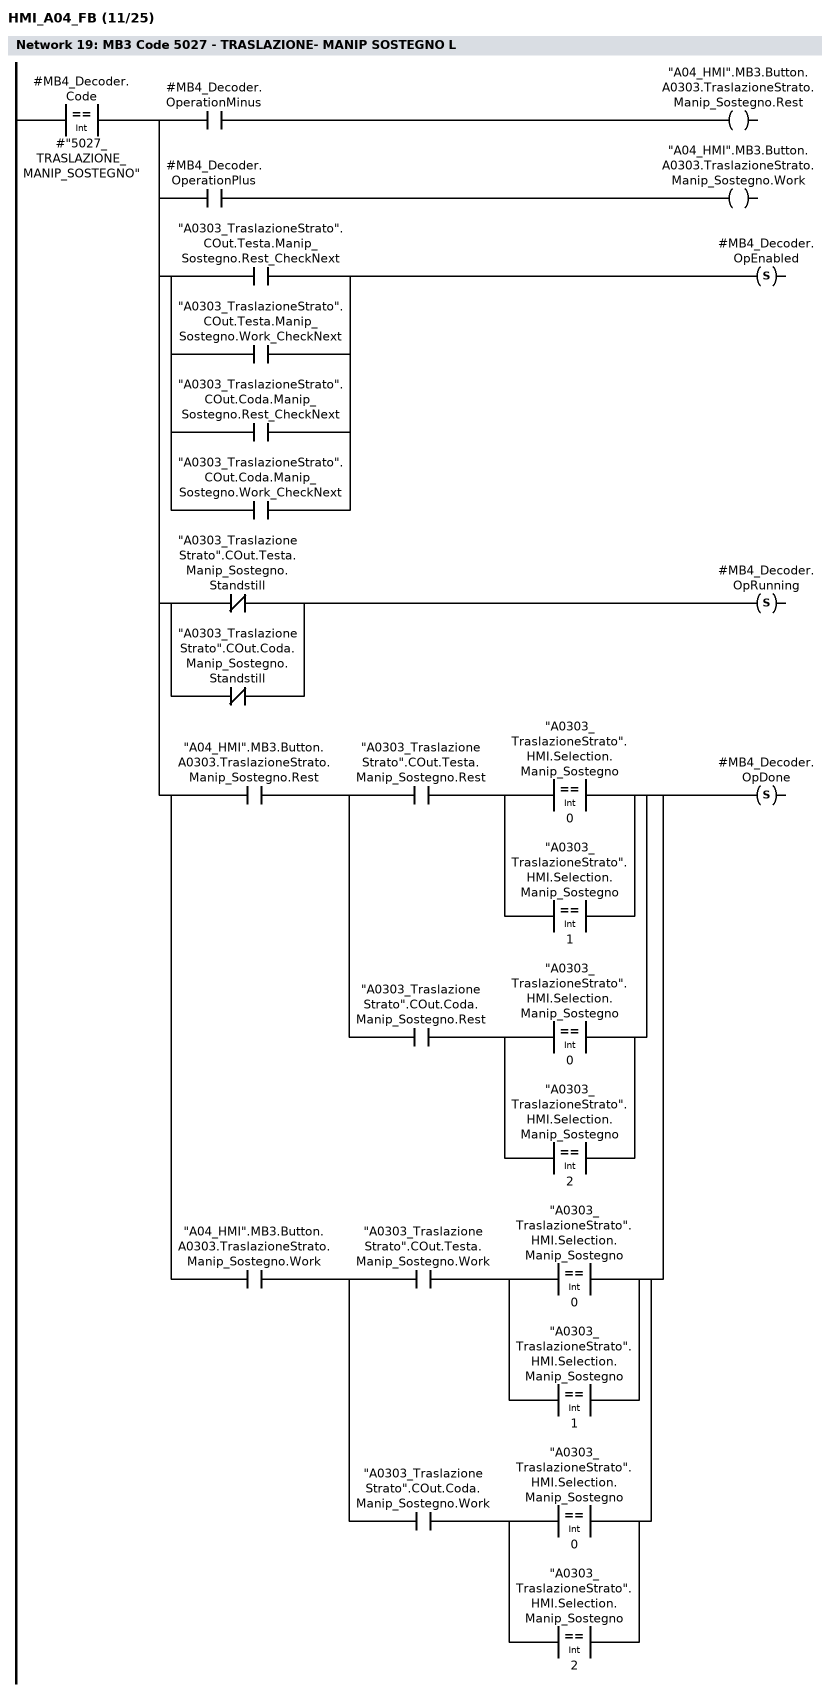
   RUNG wire#powerrail
      { S7_Templates := "SrcType := Int" } EQ_Contact(in1 := #MB4_Decoder.Code, in2 := #"5027_TRASLAZIONE_MANIP_SOSTEGNO")
      wire#w1
      Contact( #MB4_Decoder.OperationMinus )
      Coil( "A04_HMI".MB3.Button.A0303.TraslazioneStrato.Manip_Sostegno.Rest )
   END_RUNG
   RUNG wire#w1
      Contact( #MB4_Decoder.OperationPlus )
      Coil( "A04_HMI".MB3.Button.A0303.TraslazioneStrato.Manip_Sostegno.Work )
   END_RUNG
   RUNG wire#w1
      Contact( "A0303_TraslazioneStrato".COut.Testa.Manip_Sostegno.Rest_CheckNext )
      wire#w2
      S_Coil( #MB4_Decoder.OpEnabled )
   END_RUNG
   RUNG wire#w1
      Contact( "A0303_TraslazioneStrato".COut.Testa.Manip_Sostegno.Work_CheckNext )
   END_RUNG wire#w2
   RUNG wire#w1
      Contact( "A0303_TraslazioneStrato".COut.Coda.Manip_Sostegno.Rest_CheckNext )
   END_RUNG wire#w2
   RUNG wire#w1
      Contact( "A0303_TraslazioneStrato".COut.Coda.Manip_Sostegno.Work_CheckNext )
   END_RUNG wire#w2
   RUNG wire#w1
      I_Contact( "A0303_TraslazioneStrato".COut.Testa.Manip_Sostegno.Standstill )
      wire#w3
      S_Coil( #MB4_Decoder.OpRunning )
   END_RUNG
   RUNG wire#w1
      I_Contact( "A0303_TraslazioneStrato".COut.Coda.Manip_Sostegno.Standstill )
   END_RUNG wire#w3
   RUNG wire#w1
      Contact( "A04_HMI".MB3.Button.A0303.TraslazioneStrato.Manip_Sostegno.Rest )
      wire#w4
      Contact( "A0303_TraslazioneStrato".COut.Testa.Manip_Sostegno.Rest )
      wire#w5
      { S7_Templates := "SrcType := Int" } EQ_Contact(in1 := "A0303_TraslazioneStrato".HMI.Selection.Manip_Sostegno, in2 := 0)
      wire#w6
      S_Coil( #MB4_Decoder.OpDone )
   END_RUNG
   RUNG wire#w5
      { S7_Templates := "SrcType := Int" } EQ_Contact(in1 := "A0303_TraslazioneStrato".HMI.Selection.Manip_Sostegno, in2 := 1)
   END_RUNG wire#w6
   RUNG wire#w4
      Contact( "A0303_TraslazioneStrato".COut.Coda.Manip_Sostegno.Rest )
      wire#w7
      { S7_Templates := "SrcType := Int" } EQ_Contact(in1 := "A0303_TraslazioneStrato".HMI.Selection.Manip_Sostegno, in2 := 0)
   END_RUNG wire#w6
   RUNG wire#w7
      { S7_Templates := "SrcType := Int" } EQ_Contact(in1 := "A0303_TraslazioneStrato".HMI.Selection.Manip_Sostegno, in2 := 2)
   END_RUNG wire#w6
   RUNG wire#w1
      Contact( "A04_HMI".MB3.Button.A0303.TraslazioneStrato.Manip_Sostegno.Work )
      wire#w8
      Contact( "A0303_TraslazioneStrato".COut.Testa.Manip_Sostegno.Work )
      wire#w9
      { S7_Templates := "SrcType := Int" } EQ_Contact(in1 := "A0303_TraslazioneStrato".HMI.Selection.Manip_Sostegno, in2 := 0)
   END_RUNG wire#w6
   RUNG wire#w9
      { S7_Templates := "SrcType := Int" } EQ_Contact(in1 := "A0303_TraslazioneStrato".HMI.Selection.Manip_Sostegno, in2 := 1)
   END_RUNG wire#w6
   RUNG wire#w8
      Contact( "A0303_TraslazioneStrato".COut.Coda.Manip_Sostegno.Work )
      wire#w10
      { S7_Templates := "SrcType := Int" } EQ_Contact(in1 := "A0303_TraslazioneStrato".HMI.Selection.Manip_Sostegno, in2 := 0)
   END_RUNG wire#w6
   RUNG wire#w10
      { S7_Templates := "SrcType := Int" } EQ_Contact(in1 := "A0303_TraslazioneStrato".HMI.Selection.Manip_Sostegno, in2 := 2)
   END_RUNG wire#w6
   // the same network as SCL:
   #_w1 := #MB4_Decoder.Code = #"5027_TRASLAZIONE_MANIP_SOSTEGNO";
   "A04_HMI".MB3.Button.A0303.TraslazioneStrato.Manip_Sostegno.Rest := #_w1 AND #MB4_Decoder.OperationMinus;
   "A04_HMI".MB3.Button.A0303.TraslazioneStrato.Manip_Sostegno.Work := #_w1 AND #MB4_Decoder.OperationPlus;
   IF #_w1 AND ("A0303_TraslazioneStrato".COut.Testa.Manip_Sostegno.Rest_CheckNext OR "A0303_TraslazioneStrato".COut.Testa.Manip_Sostegno.Work_CheckNext OR "A0303_TraslazioneStrato".COut.Coda.Manip_Sostegno.Rest_CheckNext OR "A0303_TraslazioneStrato".COut.Coda.Manip_Sostegno.Work_CheckNext) THEN
       #MB4_Decoder.OpEnabled := TRUE;
   END_IF;
   IF #_w1 AND (NOT "A0303_TraslazioneStrato".COut.Testa.Manip_Sostegno.Standstill OR NOT "A0303_TraslazioneStrato".COut.Coda.Manip_Sostegno.Standstill) THEN
       #MB4_Decoder.OpRunning := TRUE;
   END_IF;
   IF #_w1 AND (("A04_HMI".MB3.Button.A0303.TraslazioneStrato.Manip_Sostegno.Rest AND (("A0303_TraslazioneStrato".COut.Testa.Manip_Sostegno.Rest AND (("A0303_TraslazioneStrato".HMI.Selection.Manip_Sostegno = 0) OR ("A0303_TraslazioneStrato".HMI.Selection.Manip_Sostegno = 1))) OR ("A0303_TraslazioneStrato".COut.Coda.Manip_Sostegno.Rest AND (("A0303_TraslazioneStrato".HMI.Selection.Manip_Sostegno = 0) OR ("A0303_TraslazioneStrato".HMI.Selection.Manip_Sostegno = 2))))) OR ("A04_HMI".MB3.Button.A0303.TraslazioneStrato.Manip_Sostegno.Work AND (("A0303_TraslazioneStrato".COut.Testa.Manip_Sostegno.Work AND (("A0303_TraslazioneStrato".HMI.Selection.Manip_Sostegno = 0) OR ("A0303_TraslazioneStrato".HMI.Selection.Manip_Sostegno = 1))) OR ("A0303_TraslazioneStrato".COut.Coda.Manip_Sostegno.Work AND (("A0303_TraslazioneStrato".HMI.Selection.Manip_Sostegno = 0) OR ("A0303_TraslazioneStrato".HMI.Selection.Manip_Sostegno = 2)))))) THEN
       #MB4_Decoder.OpDone := TRUE;
   END_IF;
END_REGION

REGION Network 20: MB3 Code 5028 - TRASLAZIONE- MANIP PAREGGIATORE
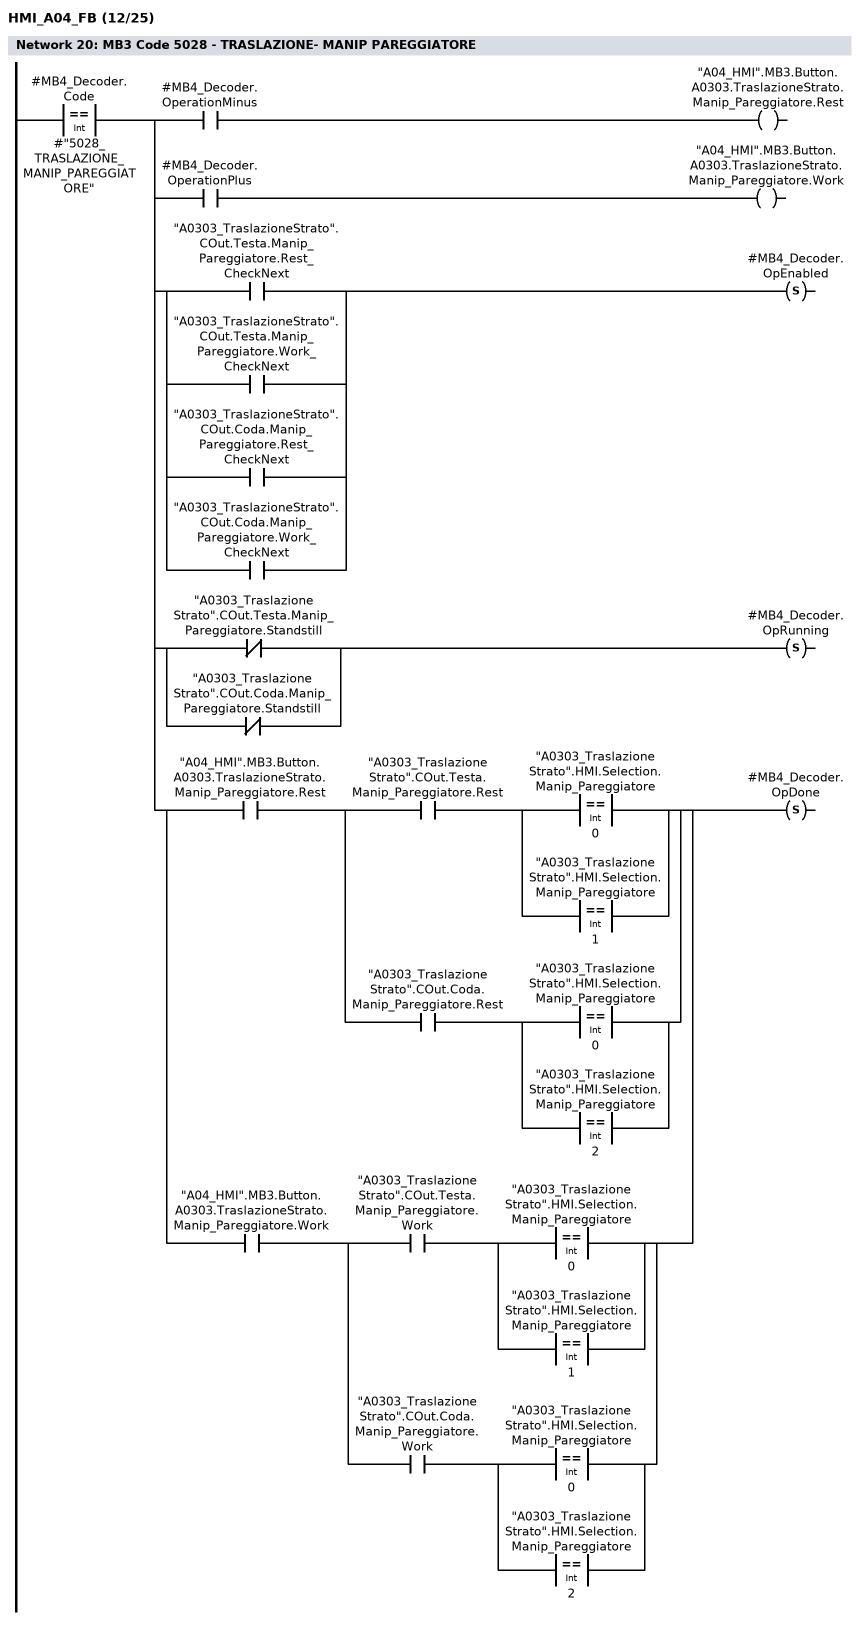
   RUNG wire#powerrail
      { S7_Templates := "SrcType := Int" } EQ_Contact(in1 := #MB4_Decoder.Code, in2 := #"5028_TRASLAZIONE_MANIP_PAREGGIATORE")
      wire#w1
      Contact( #MB4_Decoder.OperationMinus )
      Coil( "A04_HMI".MB3.Button.A0303.TraslazioneStrato.Manip_Pareggiatore.Rest )
   END_RUNG
   RUNG wire#w1
      Contact( #MB4_Decoder.OperationPlus )
      Coil( "A04_HMI".MB3.Button.A0303.TraslazioneStrato.Manip_Pareggiatore.Work )
   END_RUNG
   RUNG wire#w1
      Contact( "A0303_TraslazioneStrato".COut.Testa.Manip_Pareggiatore.Rest_CheckNext )
      wire#w2
      S_Coil( #MB4_Decoder.OpEnabled )
   END_RUNG
   RUNG wire#w1
      Contact( "A0303_TraslazioneStrato".COut.Testa.Manip_Pareggiatore.Work_CheckNext )
   END_RUNG wire#w2
   RUNG wire#w1
      Contact( "A0303_TraslazioneStrato".COut.Coda.Manip_Pareggiatore.Rest_CheckNext )
   END_RUNG wire#w2
   RUNG wire#w1
      Contact( "A0303_TraslazioneStrato".COut.Coda.Manip_Pareggiatore.Work_CheckNext )
   END_RUNG wire#w2
   RUNG wire#w1
      I_Contact( "A0303_TraslazioneStrato".COut.Testa.Manip_Pareggiatore.Standstill )
      wire#w3
      S_Coil( #MB4_Decoder.OpRunning )
   END_RUNG
   RUNG wire#w1
      I_Contact( "A0303_TraslazioneStrato".COut.Coda.Manip_Pareggiatore.Standstill )
   END_RUNG wire#w3
   RUNG wire#w1
      Contact( "A04_HMI".MB3.Button.A0303.TraslazioneStrato.Manip_Pareggiatore.Rest )
      wire#w4
      Contact( "A0303_TraslazioneStrato".COut.Testa.Manip_Pareggiatore.Rest )
      wire#w5
      { S7_Templates := "SrcType := Int" } EQ_Contact(in1 := "A0303_TraslazioneStrato".HMI.Selection.Manip_Pareggiatore, in2 := 0)
      wire#w6
      S_Coil( #MB4_Decoder.OpDone )
   END_RUNG
   RUNG wire#w5
      { S7_Templates := "SrcType := Int" } EQ_Contact(in1 := "A0303_TraslazioneStrato".HMI.Selection.Manip_Pareggiatore, in2 := 1)
   END_RUNG wire#w6
   RUNG wire#w4
      Contact( "A0303_TraslazioneStrato".COut.Coda.Manip_Pareggiatore.Rest )
      wire#w7
      { S7_Templates := "SrcType := Int" } EQ_Contact(in1 := "A0303_TraslazioneStrato".HMI.Selection.Manip_Pareggiatore, in2 := 0)
   END_RUNG wire#w6
   RUNG wire#w7
      { S7_Templates := "SrcType := Int" } EQ_Contact(in1 := "A0303_TraslazioneStrato".HMI.Selection.Manip_Pareggiatore, in2 := 2)
   END_RUNG wire#w6
   RUNG wire#w1
      Contact( "A04_HMI".MB3.Button.A0303.TraslazioneStrato.Manip_Pareggiatore.Work )
      wire#w8
      Contact( "A0303_TraslazioneStrato".COut.Testa.Manip_Pareggiatore.Work )
      wire#w9
      { S7_Templates := "SrcType := Int" } EQ_Contact(in1 := "A0303_TraslazioneStrato".HMI.Selection.Manip_Pareggiatore, in2 := 0)
   END_RUNG wire#w6
   RUNG wire#w9
      { S7_Templates := "SrcType := Int" } EQ_Contact(in1 := "A0303_TraslazioneStrato".HMI.Selection.Manip_Pareggiatore, in2 := 1)
   END_RUNG wire#w6
   RUNG wire#w8
      Contact( "A0303_TraslazioneStrato".COut.Coda.Manip_Pareggiatore.Work )
      wire#w10
      { S7_Templates := "SrcType := Int" } EQ_Contact(in1 := "A0303_TraslazioneStrato".HMI.Selection.Manip_Pareggiatore, in2 := 0)
   END_RUNG wire#w6
   RUNG wire#w10
      { S7_Templates := "SrcType := Int" } EQ_Contact(in1 := "A0303_TraslazioneStrato".HMI.Selection.Manip_Pareggiatore, in2 := 2)
   END_RUNG wire#w6
   // the same network as SCL:
   #_w1 := #MB4_Decoder.Code = #"5028_TRASLAZIONE_MANIP_PAREGGIATORE";
   "A04_HMI".MB3.Button.A0303.TraslazioneStrato.Manip_Pareggiatore.Rest := #_w1 AND #MB4_Decoder.OperationMinus;
   "A04_HMI".MB3.Button.A0303.TraslazioneStrato.Manip_Pareggiatore.Work := #_w1 AND #MB4_Decoder.OperationPlus;
   IF #_w1 AND ("A0303_TraslazioneStrato".COut.Testa.Manip_Pareggiatore.Rest_CheckNext OR "A0303_TraslazioneStrato".COut.Testa.Manip_Pareggiatore.Work_CheckNext OR "A0303_TraslazioneStrato".COut.Coda.Manip_Pareggiatore.Rest_CheckNext OR "A0303_TraslazioneStrato".COut.Coda.Manip_Pareggiatore.Work_CheckNext) THEN
       #MB4_Decoder.OpEnabled := TRUE;
   END_IF;
   IF #_w1 AND (NOT "A0303_TraslazioneStrato".COut.Testa.Manip_Pareggiatore.Standstill OR NOT "A0303_TraslazioneStrato".COut.Coda.Manip_Pareggiatore.Standstill) THEN
       #MB4_Decoder.OpRunning := TRUE;
   END_IF;
   IF #_w1 AND (("A04_HMI".MB3.Button.A0303.TraslazioneStrato.Manip_Pareggiatore.Rest AND (("A0303_TraslazioneStrato".COut.Testa.Manip_Pareggiatore.Rest AND (("A0303_TraslazioneStrato".HMI.Selection.Manip_Pareggiatore = 0) OR ("A0303_TraslazioneStrato".HMI.Selection.Manip_Pareggiatore = 1))) OR ("A0303_TraslazioneStrato".COut.Coda.Manip_Pareggiatore.Rest AND (("A0303_TraslazioneStrato".HMI.Selection.Manip_Pareggiatore = 0) OR ("A0303_TraslazioneStrato".HMI.Selection.Manip_Pareggiatore = 2))))) OR ("A04_HMI".MB3.Button.A0303.TraslazioneStrato.Manip_Pareggiatore.Work AND (("A0303_TraslazioneStrato".COut.Testa.Manip_Pareggiatore.Work AND (("A0303_TraslazioneStrato".HMI.Selection.Manip_Pareggiatore = 0) OR ("A0303_TraslazioneStrato".HMI.Selection.Manip_Pareggiatore = 1))) OR ("A0303_TraslazioneStrato".COut.Coda.Manip_Pareggiatore.Work AND (("A0303_TraslazioneStrato".HMI.Selection.Manip_Pareggiatore = 0) OR ("A0303_TraslazioneStrato".HMI.Selection.Manip_Pareggiatore = 2)))))) THEN
       #MB4_Decoder.OpDone := TRUE;
   END_IF;
END_REGION

REGION Network 21: MB3 Code 5029 - TRASLAZIONE- SOSTEGNO VERTICALE
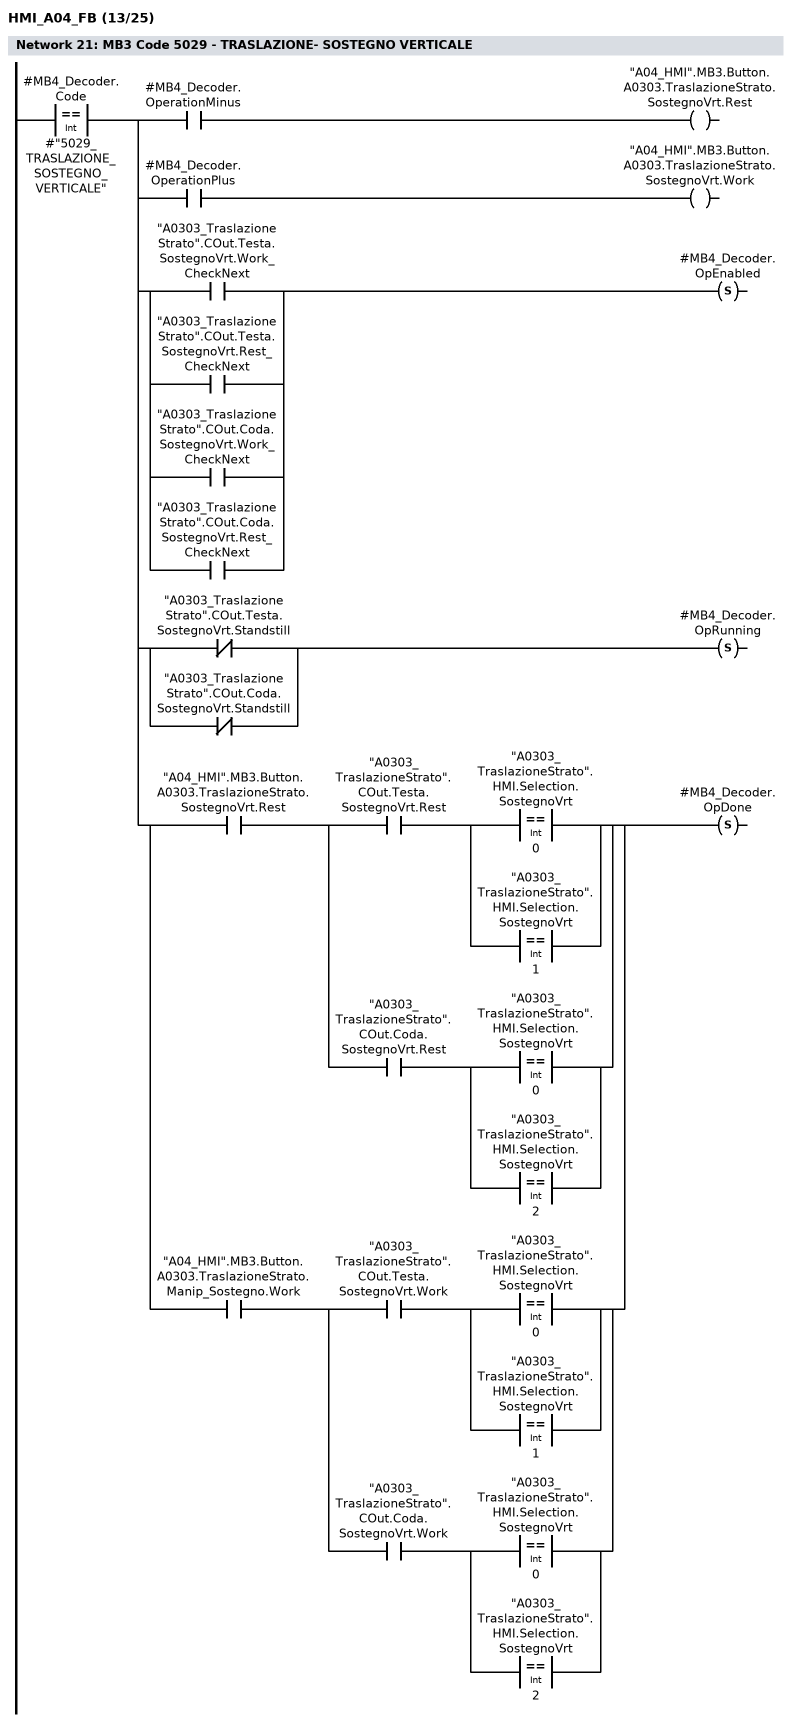
   RUNG wire#powerrail
      { S7_Templates := "SrcType := Int" } EQ_Contact(in1 := #MB4_Decoder.Code, in2 := #"5029_TRASLAZIONE_SOSTEGNO_VERTICALE")
      wire#w1
      Contact( #MB4_Decoder.OperationMinus )
      Coil( "A04_HMI".MB3.Button.A0303.TraslazioneStrato.SostegnoVrt.Rest )
   END_RUNG
   RUNG wire#w1
      Contact( #MB4_Decoder.OperationPlus )
      Coil( "A04_HMI".MB3.Button.A0303.TraslazioneStrato.SostegnoVrt.Work )
   END_RUNG
   RUNG wire#w1
      Contact( "A0303_TraslazioneStrato".COut.Testa.SostegnoVrt.Work_CheckNext )
      wire#w2
      S_Coil( #MB4_Decoder.OpEnabled )
   END_RUNG
   RUNG wire#w1
      Contact( "A0303_TraslazioneStrato".COut.Testa.SostegnoVrt.Rest_CheckNext )
   END_RUNG wire#w2
   RUNG wire#w1
      Contact( "A0303_TraslazioneStrato".COut.Coda.SostegnoVrt.Work_CheckNext )
   END_RUNG wire#w2
   RUNG wire#w1
      Contact( "A0303_TraslazioneStrato".COut.Coda.SostegnoVrt.Rest_CheckNext )
   END_RUNG wire#w2
   RUNG wire#w1
      I_Contact( "A0303_TraslazioneStrato".COut.Testa.SostegnoVrt.Standstill )
      wire#w3
      S_Coil( #MB4_Decoder.OpRunning )
   END_RUNG
   RUNG wire#w1
      I_Contact( "A0303_TraslazioneStrato".COut.Coda.SostegnoVrt.Standstill )
   END_RUNG wire#w3
   RUNG wire#w1
      Contact( "A04_HMI".MB3.Button.A0303.TraslazioneStrato.SostegnoVrt.Rest )
      wire#w4
      Contact( "A0303_TraslazioneStrato".COut.Testa.SostegnoVrt.Rest )
      wire#w5
      { S7_Templates := "SrcType := Int" } EQ_Contact(in1 := "A0303_TraslazioneStrato".HMI.Selection.SostegnoVrt, in2 := 0)
      wire#w6
      S_Coil( #MB4_Decoder.OpDone )
   END_RUNG
   RUNG wire#w5
      { S7_Templates := "SrcType := Int" } EQ_Contact(in1 := "A0303_TraslazioneStrato".HMI.Selection.SostegnoVrt, in2 := 1)
   END_RUNG wire#w6
   RUNG wire#w4
      Contact( "A0303_TraslazioneStrato".COut.Coda.SostegnoVrt.Rest )
      wire#w7
      { S7_Templates := "SrcType := Int" } EQ_Contact(in1 := "A0303_TraslazioneStrato".HMI.Selection.SostegnoVrt, in2 := 0)
   END_RUNG wire#w6
   RUNG wire#w7
      { S7_Templates := "SrcType := Int" } EQ_Contact(in1 := "A0303_TraslazioneStrato".HMI.Selection.SostegnoVrt, in2 := 2)
   END_RUNG wire#w6
   RUNG wire#w1
      Contact( "A04_HMI".MB3.Button.A0303.TraslazioneStrato.Manip_Sostegno.Work )
      wire#w8
      Contact( "A0303_TraslazioneStrato".COut.Testa.SostegnoVrt.Work )
      wire#w9
      { S7_Templates := "SrcType := Int" } EQ_Contact(in1 := "A0303_TraslazioneStrato".HMI.Selection.SostegnoVrt, in2 := 0)
   END_RUNG wire#w6
   RUNG wire#w9
      { S7_Templates := "SrcType := Int" } EQ_Contact(in1 := "A0303_TraslazioneStrato".HMI.Selection.SostegnoVrt, in2 := 1)
   END_RUNG wire#w6
   RUNG wire#w8
      Contact( "A0303_TraslazioneStrato".COut.Coda.SostegnoVrt.Work )
      wire#w10
      { S7_Templates := "SrcType := Int" } EQ_Contact(in1 := "A0303_TraslazioneStrato".HMI.Selection.SostegnoVrt, in2 := 0)
   END_RUNG wire#w6
   RUNG wire#w10
      { S7_Templates := "SrcType := Int" } EQ_Contact(in1 := "A0303_TraslazioneStrato".HMI.Selection.SostegnoVrt, in2 := 2)
   END_RUNG wire#w6
   // the same network as SCL:
   #_w1 := #MB4_Decoder.Code = #"5029_TRASLAZIONE_SOSTEGNO_VERTICALE";
   "A04_HMI".MB3.Button.A0303.TraslazioneStrato.SostegnoVrt.Rest := #_w1 AND #MB4_Decoder.OperationMinus;
   "A04_HMI".MB3.Button.A0303.TraslazioneStrato.SostegnoVrt.Work := #_w1 AND #MB4_Decoder.OperationPlus;
   IF #_w1 AND ("A0303_TraslazioneStrato".COut.Testa.SostegnoVrt.Work_CheckNext OR "A0303_TraslazioneStrato".COut.Testa.SostegnoVrt.Rest_CheckNext OR "A0303_TraslazioneStrato".COut.Coda.SostegnoVrt.Work_CheckNext OR "A0303_TraslazioneStrato".COut.Coda.SostegnoVrt.Rest_CheckNext) THEN
       #MB4_Decoder.OpEnabled := TRUE;
   END_IF;
   IF #_w1 AND (NOT "A0303_TraslazioneStrato".COut.Testa.SostegnoVrt.Standstill OR NOT "A0303_TraslazioneStrato".COut.Coda.SostegnoVrt.Standstill) THEN
       #MB4_Decoder.OpRunning := TRUE;
   END_IF;
   IF #_w1 AND (("A04_HMI".MB3.Button.A0303.TraslazioneStrato.SostegnoVrt.Rest AND (("A0303_TraslazioneStrato".COut.Testa.SostegnoVrt.Rest AND (("A0303_TraslazioneStrato".HMI.Selection.SostegnoVrt = 0) OR ("A0303_TraslazioneStrato".HMI.Selection.SostegnoVrt = 1))) OR ("A0303_TraslazioneStrato".COut.Coda.SostegnoVrt.Rest AND (("A0303_TraslazioneStrato".HMI.Selection.SostegnoVrt = 0) OR ("A0303_TraslazioneStrato".HMI.Selection.SostegnoVrt = 2))))) OR ("A04_HMI".MB3.Button.A0303.TraslazioneStrato.Manip_Sostegno.Work AND (("A0303_TraslazioneStrato".COut.Testa.SostegnoVrt.Work AND (("A0303_TraslazioneStrato".HMI.Selection.SostegnoVrt = 0) OR ("A0303_TraslazioneStrato".HMI.Selection.SostegnoVrt = 1))) OR ("A0303_TraslazioneStrato".COut.Coda.SostegnoVrt.Work AND (("A0303_TraslazioneStrato".HMI.Selection.SostegnoVrt = 0) OR ("A0303_TraslazioneStrato".HMI.Selection.SostegnoVrt = 2)))))) THEN
       #MB4_Decoder.OpDone := TRUE;
   END_IF;
END_REGION

REGION Network 22: MB3 Code 5031- SOLLEVAMENTO - OP
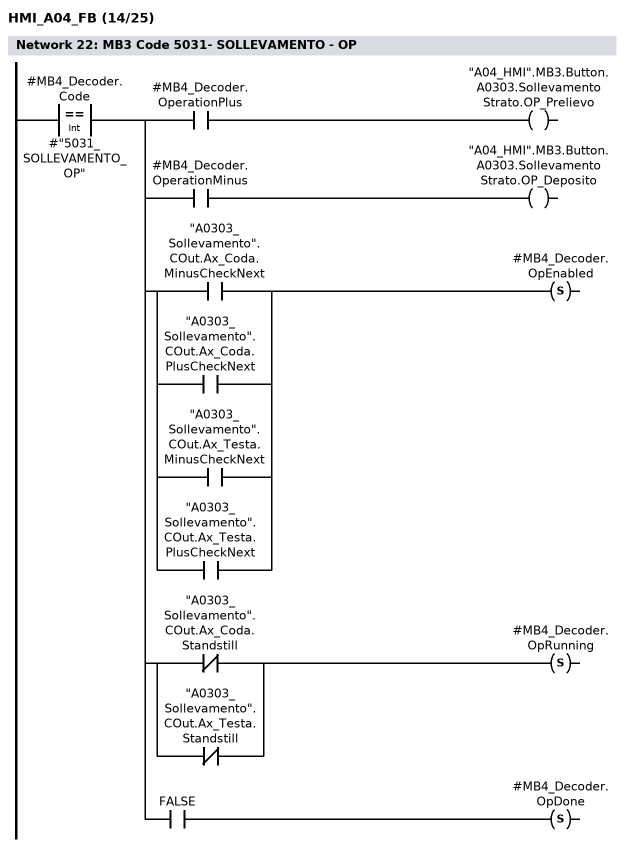
   RUNG wire#powerrail
      { S7_Templates := "SrcType := Int" } EQ_Contact(in1 := #MB4_Decoder.Code, in2 := #"5031_SOLLEVAMENTO_OP")
      wire#w1
      Contact( #MB4_Decoder.OperationPlus )
      Coil( "A04_HMI".MB3.Button.A0303.SollevamentoStrato.OP_Prelievo )
   END_RUNG
   RUNG wire#w1
      Contact( #MB4_Decoder.OperationMinus )
      Coil( "A04_HMI".MB3.Button.A0303.SollevamentoStrato.OP_Deposito )
   END_RUNG
   RUNG wire#w1
      Contact( "A0303_Sollevamento".COut.Ax_Coda.MinusCheckNext )
      wire#w2
      S_Coil( #MB4_Decoder.OpEnabled )
   END_RUNG
   RUNG wire#w1
      Contact( "A0303_Sollevamento".COut.Ax_Coda.PlusCheckNext )
   END_RUNG wire#w2
   RUNG wire#w1
      Contact( "A0303_Sollevamento".COut.Ax_Testa.MinusCheckNext )
   END_RUNG wire#w2
   RUNG wire#w1
      Contact( "A0303_Sollevamento".COut.Ax_Testa.PlusCheckNext )
   END_RUNG wire#w2
   RUNG wire#w1
      I_Contact( "A0303_Sollevamento".COut.Ax_Coda.Standstill )
      wire#w3
      S_Coil( #MB4_Decoder.OpRunning )
   END_RUNG
   RUNG wire#w1
      I_Contact( "A0303_Sollevamento".COut.Ax_Testa.Standstill )
   END_RUNG wire#w3
   RUNG wire#w1
      Contact( FALSE )
      S_Coil( #MB4_Decoder.OpDone )
   END_RUNG
   // the same network as SCL:
   #_w1 := #MB4_Decoder.Code = #"5031_SOLLEVAMENTO_OP";
   "A04_HMI".MB3.Button.A0303.SollevamentoStrato.OP_Prelievo := #_w1 AND #MB4_Decoder.OperationPlus;
   "A04_HMI".MB3.Button.A0303.SollevamentoStrato.OP_Deposito := #_w1 AND #MB4_Decoder.OperationMinus;
   IF #_w1 AND ("A0303_Sollevamento".COut.Ax_Coda.MinusCheckNext OR "A0303_Sollevamento".COut.Ax_Coda.PlusCheckNext OR "A0303_Sollevamento".COut.Ax_Testa.MinusCheckNext OR "A0303_Sollevamento".COut.Ax_Testa.PlusCheckNext) THEN
       #MB4_Decoder.OpEnabled := TRUE;
   END_IF;
   IF #_w1 AND (NOT "A0303_Sollevamento".COut.Ax_Coda.Standstill OR NOT "A0303_Sollevamento".COut.Ax_Testa.Standstill) THEN
       #MB4_Decoder.OpRunning := TRUE;
   END_IF;
   IF #_w1 AND FALSE THEN #MB4_Decoder.OpDone := TRUE; END_IF;
END_REGION

REGION Network 23: MB3 Code 5032- SOLLEVAMENTO - AX - JOG
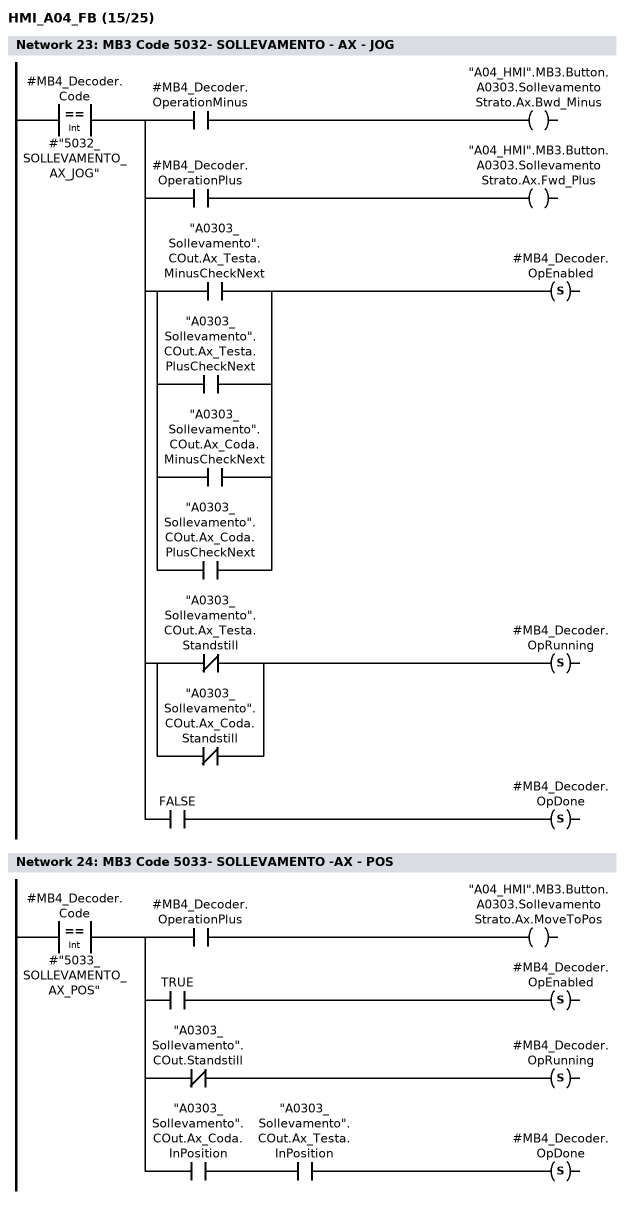
   RUNG wire#powerrail
      { S7_Templates := "SrcType := Int" } EQ_Contact(in1 := #MB4_Decoder.Code, in2 := #"5032_SOLLEVAMENTO_AX_JOG")
      wire#w1
      Contact( #MB4_Decoder.OperationMinus )
      Coil( "A04_HMI".MB3.Button.A0303.SollevamentoStrato.Ax.Bwd_Minus )
   END_RUNG
   RUNG wire#w1
      Contact( #MB4_Decoder.OperationPlus )
      Coil( "A04_HMI".MB3.Button.A0303.SollevamentoStrato.Ax.Fwd_Plus )
   END_RUNG
   RUNG wire#w1
      Contact( "A0303_Sollevamento".COut.Ax_Testa.MinusCheckNext )
      wire#w2
      S_Coil( #MB4_Decoder.OpEnabled )
   END_RUNG
   RUNG wire#w1
      Contact( "A0303_Sollevamento".COut.Ax_Testa.PlusCheckNext )
   END_RUNG wire#w2
   RUNG wire#w1
      Contact( "A0303_Sollevamento".COut.Ax_Coda.MinusCheckNext )
   END_RUNG wire#w2
   RUNG wire#w1
      Contact( "A0303_Sollevamento".COut.Ax_Coda.PlusCheckNext )
   END_RUNG wire#w2
   RUNG wire#w1
      I_Contact( "A0303_Sollevamento".COut.Ax_Testa.Standstill )
      wire#w3
      S_Coil( #MB4_Decoder.OpRunning )
   END_RUNG
   RUNG wire#w1
      I_Contact( "A0303_Sollevamento".COut.Ax_Coda.Standstill )
   END_RUNG wire#w3
   RUNG wire#w1
      Contact( FALSE )
      S_Coil( #MB4_Decoder.OpDone )
   END_RUNG
   // the same network as SCL:
   #_w1 := #MB4_Decoder.Code = #"5032_SOLLEVAMENTO_AX_JOG";
   "A04_HMI".MB3.Button.A0303.SollevamentoStrato.Ax.Bwd_Minus := #_w1 AND #MB4_Decoder.OperationMinus;
   "A04_HMI".MB3.Button.A0303.SollevamentoStrato.Ax.Fwd_Plus := #_w1 AND #MB4_Decoder.OperationPlus;
   IF #_w1 AND ("A0303_Sollevamento".COut.Ax_Testa.MinusCheckNext OR "A0303_Sollevamento".COut.Ax_Testa.PlusCheckNext OR "A0303_Sollevamento".COut.Ax_Coda.MinusCheckNext OR "A0303_Sollevamento".COut.Ax_Coda.PlusCheckNext) THEN
       #MB4_Decoder.OpEnabled := TRUE;
   END_IF;
   IF #_w1 AND (NOT "A0303_Sollevamento".COut.Ax_Testa.Standstill OR NOT "A0303_Sollevamento".COut.Ax_Coda.Standstill) THEN
       #MB4_Decoder.OpRunning := TRUE;
   END_IF;
   IF #_w1 AND FALSE THEN #MB4_Decoder.OpDone := TRUE; END_IF;
END_REGION

REGION Network 24: MB3 Code 5033- SOLLEVAMENTO -AX - POS
   RUNG wire#powerrail
      { S7_Templates := "SrcType := Int" } EQ_Contact(in1 := #MB4_Decoder.Code, in2 := #"5033_SOLLEVAMENTO_AX_POS")
      wire#w1
      Contact( #MB4_Decoder.OperationPlus )
      Coil( "A04_HMI".MB3.Button.A0303.SollevamentoStrato.Ax.MoveToPos )
   END_RUNG
   RUNG wire#w1
      Contact( TRUE )
      S_Coil( #MB4_Decoder.OpEnabled )
   END_RUNG
   RUNG wire#w1
      I_Contact( "A0303_Sollevamento".COut.Standstill )
      S_Coil( #MB4_Decoder.OpRunning )
   END_RUNG
   RUNG wire#w1
      Contact( "A0303_Sollevamento".COut.Ax_Coda.InPosition )
      Contact( "A0303_Sollevamento".COut.Ax_Testa.InPosition )
      S_Coil( #MB4_Decoder.OpDone )
   END_RUNG
   // the same network as SCL:
   #_w1 := #MB4_Decoder.Code = #"5033_SOLLEVAMENTO_AX_POS";
   "A04_HMI".MB3.Button.A0303.SollevamentoStrato.Ax.MoveToPos := #_w1 AND #MB4_Decoder.OperationPlus;
   IF #_w1 AND TRUE THEN #MB4_Decoder.OpEnabled := TRUE; END_IF;
   IF #_w1 AND NOT "A0303_Sollevamento".COut.Standstill THEN #MB4_Decoder.OpRunning := TRUE; END_IF;
   IF #_w1 AND "A0303_Sollevamento".COut.Ax_Coda.InPosition AND "A0303_Sollevamento".COut.Ax_Testa.InPosition THEN
       #MB4_Decoder.OpDone := TRUE;
   END_IF;
END_REGION

REGION Network 25: MB3 Code 5041- SOSTEGNO ANTIRIBALTAMENTO - OP
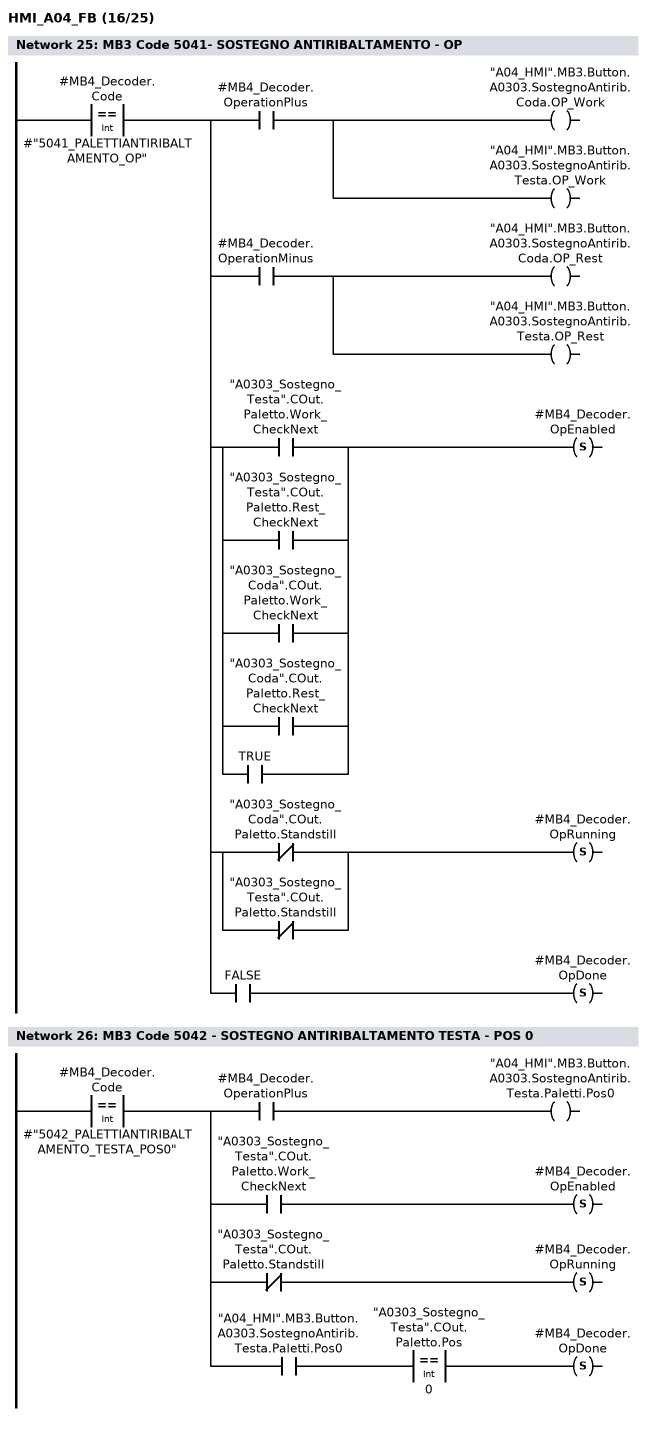
   RUNG wire#powerrail
      { S7_Templates := "SrcType := Int" } EQ_Contact(in1 := #MB4_Decoder.Code, in2 := #"5041_PALETTIANTIRIBALTAMENTO_OP")
      wire#w1
      Contact( #MB4_Decoder.OperationPlus )
      wire#w2
      Coil( "A04_HMI".MB3.Button.A0303.SostegnoAntirib.Coda.OP_Work )
   END_RUNG
   RUNG wire#w2
      Coil( "A04_HMI".MB3.Button.A0303.SostegnoAntirib.Testa.OP_Work )
   END_RUNG
   RUNG wire#w1
      Contact( #MB4_Decoder.OperationMinus )
      wire#w3
      Coil( "A04_HMI".MB3.Button.A0303.SostegnoAntirib.Coda.OP_Rest )
   END_RUNG
   RUNG wire#w3
      Coil( "A04_HMI".MB3.Button.A0303.SostegnoAntirib.Testa.OP_Rest )
   END_RUNG
   RUNG wire#w1
      Contact( "A0303_Sostegno_Testa".COut.Paletto.Work_CheckNext )
      wire#w4
      S_Coil( #MB4_Decoder.OpEnabled )
   END_RUNG
   RUNG wire#w1
      Contact( "A0303_Sostegno_Testa".COut.Paletto.Rest_CheckNext )
   END_RUNG wire#w4
   RUNG wire#w1
      Contact( "A0303_Sostegno_Coda".COut.Paletto.Work_CheckNext )
   END_RUNG wire#w4
   RUNG wire#w1
      Contact( "A0303_Sostegno_Coda".COut.Paletto.Rest_CheckNext )
   END_RUNG wire#w4
   RUNG wire#w1
      Contact( TRUE )
   END_RUNG wire#w4
   RUNG wire#w1
      I_Contact( "A0303_Sostegno_Coda".COut.Paletto.Standstill )
      wire#w5
      S_Coil( #MB4_Decoder.OpRunning )
   END_RUNG
   RUNG wire#w1
      I_Contact( "A0303_Sostegno_Testa".COut.Paletto.Standstill )
   END_RUNG wire#w5
   RUNG wire#w1
      Contact( FALSE )
      S_Coil( #MB4_Decoder.OpDone )
   END_RUNG
   // the same network as SCL:
   #_w1 := #MB4_Decoder.Code = #"5041_PALETTIANTIRIBALTAMENTO_OP";
   "A04_HMI".MB3.Button.A0303.SostegnoAntirib.Coda.OP_Work := #_w1 AND #MB4_Decoder.OperationPlus;
   "A04_HMI".MB3.Button.A0303.SostegnoAntirib.Testa.OP_Work := "A04_HMI".MB3.Button.A0303.SostegnoAntirib.Coda.OP_Work;
   "A04_HMI".MB3.Button.A0303.SostegnoAntirib.Coda.OP_Rest := #_w1 AND #MB4_Decoder.OperationMinus;
   "A04_HMI".MB3.Button.A0303.SostegnoAntirib.Testa.OP_Rest := "A04_HMI".MB3.Button.A0303.SostegnoAntirib.Coda.OP_Rest;
   IF #_w1 AND ("A0303_Sostegno_Testa".COut.Paletto.Work_CheckNext OR "A0303_Sostegno_Testa".COut.Paletto.Rest_CheckNext OR "A0303_Sostegno_Coda".COut.Paletto.Work_CheckNext OR "A0303_Sostegno_Coda".COut.Paletto.Rest_CheckNext OR TRUE) THEN
       #MB4_Decoder.OpEnabled := TRUE;
   END_IF;
   IF #_w1 AND (NOT "A0303_Sostegno_Coda".COut.Paletto.Standstill OR NOT "A0303_Sostegno_Testa".COut.Paletto.Standstill) THEN
       #MB4_Decoder.OpRunning := TRUE;
   END_IF;
   IF #_w1 AND FALSE THEN #MB4_Decoder.OpDone := TRUE; END_IF;
END_REGION

REGION Network 26: MB3 Code 5042 - SOSTEGNO ANTIRIBALTAMENTO TESTA - POS 0
   RUNG wire#powerrail
      { S7_Templates := "SrcType := Int" } EQ_Contact(in1 := #MB4_Decoder.Code, in2 := #"5042_PALETTIANTIRIBALTAMENTO_TESTA_POS0")
      wire#w1
      Contact( #MB4_Decoder.OperationPlus )
      Coil( "A04_HMI".MB3.Button.A0303.SostegnoAntirib.Testa.Paletti.Pos0 )
   END_RUNG
   RUNG wire#w1
      Contact( "A0303_Sostegno_Testa".COut.Paletto.Work_CheckNext )
      S_Coil( #MB4_Decoder.OpEnabled )
   END_RUNG
   RUNG wire#w1
      I_Contact( "A0303_Sostegno_Testa".COut.Paletto.Standstill )
      S_Coil( #MB4_Decoder.OpRunning )
   END_RUNG
   RUNG wire#w1
      Contact( "A04_HMI".MB3.Button.A0303.SostegnoAntirib.Testa.Paletti.Pos0 )
      { S7_Templates := "SrcType := Int" } EQ_Contact(in1 := "A0303_Sostegno_Testa".COut.Paletto.Pos, in2 := 0)
      S_Coil( #MB4_Decoder.OpDone )
   END_RUNG
   // the same network as SCL:
   #_w1 := #MB4_Decoder.Code = #"5042_PALETTIANTIRIBALTAMENTO_TESTA_POS0";
   "A04_HMI".MB3.Button.A0303.SostegnoAntirib.Testa.Paletti.Pos0 := #_w1 AND #MB4_Decoder.OperationPlus;
   IF #_w1 AND "A0303_Sostegno_Testa".COut.Paletto.Work_CheckNext THEN
       #MB4_Decoder.OpEnabled := TRUE;
   END_IF;
   IF #_w1 AND NOT "A0303_Sostegno_Testa".COut.Paletto.Standstill THEN
       #MB4_Decoder.OpRunning := TRUE;
   END_IF;
   IF #_w1 AND "A04_HMI".MB3.Button.A0303.SostegnoAntirib.Testa.Paletti.Pos0 AND ("A0303_Sostegno_Testa".COut.Paletto.Pos = 0) THEN
       #MB4_Decoder.OpDone := TRUE;
   END_IF;
END_REGION

REGION Network 27: MB3 Code 5043 - SOSTEGNO ANTIRIBALTAMENTO TESTA - POS 1
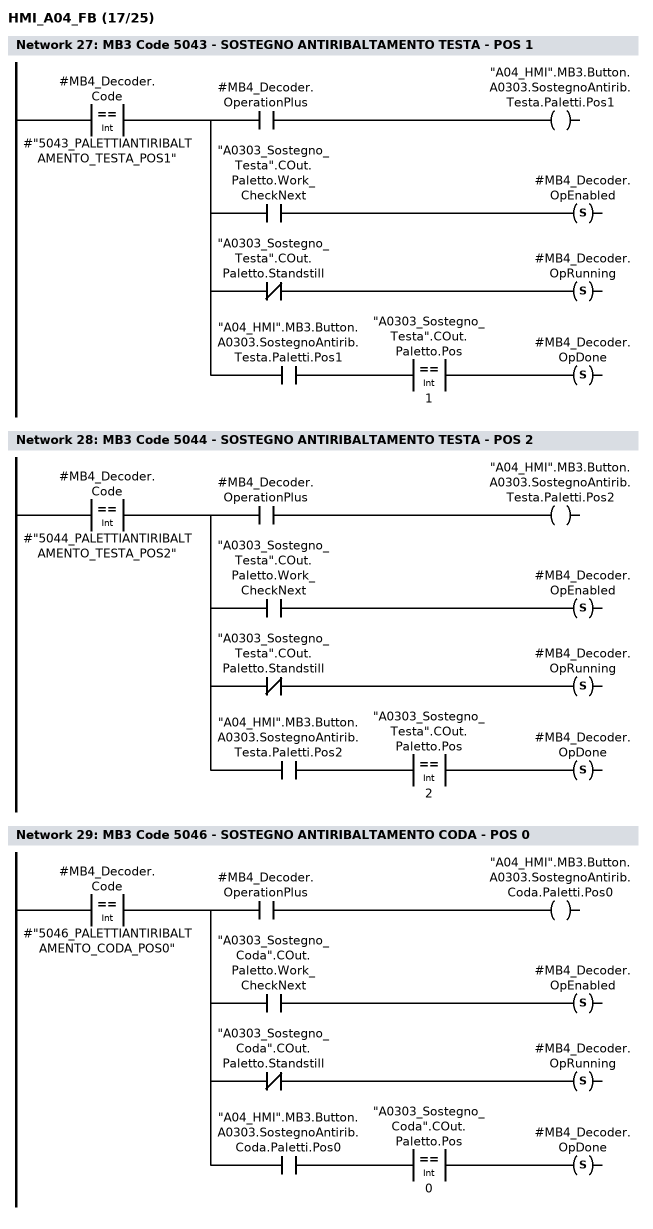
   RUNG wire#powerrail
      { S7_Templates := "SrcType := Int" } EQ_Contact(in1 := #MB4_Decoder.Code, in2 := #"5043_PALETTIANTIRIBALTAMENTO_TESTA_POS1")
      wire#w1
      Contact( #MB4_Decoder.OperationPlus )
      Coil( "A04_HMI".MB3.Button.A0303.SostegnoAntirib.Testa.Paletti.Pos1 )
   END_RUNG
   RUNG wire#w1
      Contact( "A0303_Sostegno_Testa".COut.Paletto.Work_CheckNext )
      S_Coil( #MB4_Decoder.OpEnabled )
   END_RUNG
   RUNG wire#w1
      I_Contact( "A0303_Sostegno_Testa".COut.Paletto.Standstill )
      S_Coil( #MB4_Decoder.OpRunning )
   END_RUNG
   RUNG wire#w1
      Contact( "A04_HMI".MB3.Button.A0303.SostegnoAntirib.Testa.Paletti.Pos1 )
      { S7_Templates := "SrcType := Int" } EQ_Contact(in1 := "A0303_Sostegno_Testa".COut.Paletto.Pos, in2 := 1)
      S_Coil( #MB4_Decoder.OpDone )
   END_RUNG
   // the same network as SCL:
   #_w1 := #MB4_Decoder.Code = #"5043_PALETTIANTIRIBALTAMENTO_TESTA_POS1";
   "A04_HMI".MB3.Button.A0303.SostegnoAntirib.Testa.Paletti.Pos1 := #_w1 AND #MB4_Decoder.OperationPlus;
   IF #_w1 AND "A0303_Sostegno_Testa".COut.Paletto.Work_CheckNext THEN
       #MB4_Decoder.OpEnabled := TRUE;
   END_IF;
   IF #_w1 AND NOT "A0303_Sostegno_Testa".COut.Paletto.Standstill THEN
       #MB4_Decoder.OpRunning := TRUE;
   END_IF;
   IF #_w1 AND "A04_HMI".MB3.Button.A0303.SostegnoAntirib.Testa.Paletti.Pos1 AND ("A0303_Sostegno_Testa".COut.Paletto.Pos = 1) THEN
       #MB4_Decoder.OpDone := TRUE;
   END_IF;
END_REGION

REGION Network 28: MB3 Code 5044 - SOSTEGNO ANTIRIBALTAMENTO TESTA - POS 2
   RUNG wire#powerrail
      { S7_Templates := "SrcType := Int" } EQ_Contact(in1 := #MB4_Decoder.Code, in2 := #"5044_PALETTIANTIRIBALTAMENTO_TESTA_POS2")
      wire#w1
      Contact( #MB4_Decoder.OperationPlus )
      Coil( "A04_HMI".MB3.Button.A0303.SostegnoAntirib.Testa.Paletti.Pos2 )
   END_RUNG
   RUNG wire#w1
      Contact( "A0303_Sostegno_Testa".COut.Paletto.Work_CheckNext )
      S_Coil( #MB4_Decoder.OpEnabled )
   END_RUNG
   RUNG wire#w1
      I_Contact( "A0303_Sostegno_Testa".COut.Paletto.Standstill )
      S_Coil( #MB4_Decoder.OpRunning )
   END_RUNG
   RUNG wire#w1
      Contact( "A04_HMI".MB3.Button.A0303.SostegnoAntirib.Testa.Paletti.Pos2 )
      { S7_Templates := "SrcType := Int" } EQ_Contact(in1 := "A0303_Sostegno_Testa".COut.Paletto.Pos, in2 := 2)
      S_Coil( #MB4_Decoder.OpDone )
   END_RUNG
   // the same network as SCL:
   #_w1 := #MB4_Decoder.Code = #"5044_PALETTIANTIRIBALTAMENTO_TESTA_POS2";
   "A04_HMI".MB3.Button.A0303.SostegnoAntirib.Testa.Paletti.Pos2 := #_w1 AND #MB4_Decoder.OperationPlus;
   IF #_w1 AND "A0303_Sostegno_Testa".COut.Paletto.Work_CheckNext THEN
       #MB4_Decoder.OpEnabled := TRUE;
   END_IF;
   IF #_w1 AND NOT "A0303_Sostegno_Testa".COut.Paletto.Standstill THEN
       #MB4_Decoder.OpRunning := TRUE;
   END_IF;
   IF #_w1 AND "A04_HMI".MB3.Button.A0303.SostegnoAntirib.Testa.Paletti.Pos2 AND ("A0303_Sostegno_Testa".COut.Paletto.Pos = 2) THEN
       #MB4_Decoder.OpDone := TRUE;
   END_IF;
END_REGION

REGION Network 29: MB3 Code 5046 - SOSTEGNO ANTIRIBALTAMENTO CODA - POS 0
   RUNG wire#powerrail
      { S7_Templates := "SrcType := Int" } EQ_Contact(in1 := #MB4_Decoder.Code, in2 := #"5046_PALETTIANTIRIBALTAMENTO_CODA_POS0")
      wire#w1
      Contact( #MB4_Decoder.OperationPlus )
      Coil( "A04_HMI".MB3.Button.A0303.SostegnoAntirib.Coda.Paletti.Pos0 )
   END_RUNG
   RUNG wire#w1
      Contact( "A0303_Sostegno_Coda".COut.Paletto.Work_CheckNext )
      S_Coil( #MB4_Decoder.OpEnabled )
   END_RUNG
   RUNG wire#w1
      I_Contact( "A0303_Sostegno_Coda".COut.Paletto.Standstill )
      S_Coil( #MB4_Decoder.OpRunning )
   END_RUNG
   RUNG wire#w1
      Contact( "A04_HMI".MB3.Button.A0303.SostegnoAntirib.Coda.Paletti.Pos0 )
      { S7_Templates := "SrcType := Int" } EQ_Contact(in1 := "A0303_Sostegno_Coda".COut.Paletto.Pos, in2 := 0)
      S_Coil( #MB4_Decoder.OpDone )
   END_RUNG
   // the same network as SCL:
   #_w1 := #MB4_Decoder.Code = #"5046_PALETTIANTIRIBALTAMENTO_CODA_POS0";
   "A04_HMI".MB3.Button.A0303.SostegnoAntirib.Coda.Paletti.Pos0 := #_w1 AND #MB4_Decoder.OperationPlus;
   IF #_w1 AND "A0303_Sostegno_Coda".COut.Paletto.Work_CheckNext THEN #MB4_Decoder.OpEnabled := TRUE; END_IF;
   IF #_w1 AND NOT "A0303_Sostegno_Coda".COut.Paletto.Standstill THEN #MB4_Decoder.OpRunning := TRUE; END_IF;
   IF #_w1 AND "A04_HMI".MB3.Button.A0303.SostegnoAntirib.Coda.Paletti.Pos0 AND ("A0303_Sostegno_Coda".COut.Paletto.Pos = 0) THEN
       #MB4_Decoder.OpDone := TRUE;
   END_IF;
END_REGION

REGION Network 30: MB3 Code 5047 - SOSTEGNO ANTIRIBALTAMENTO CODA - POS 1
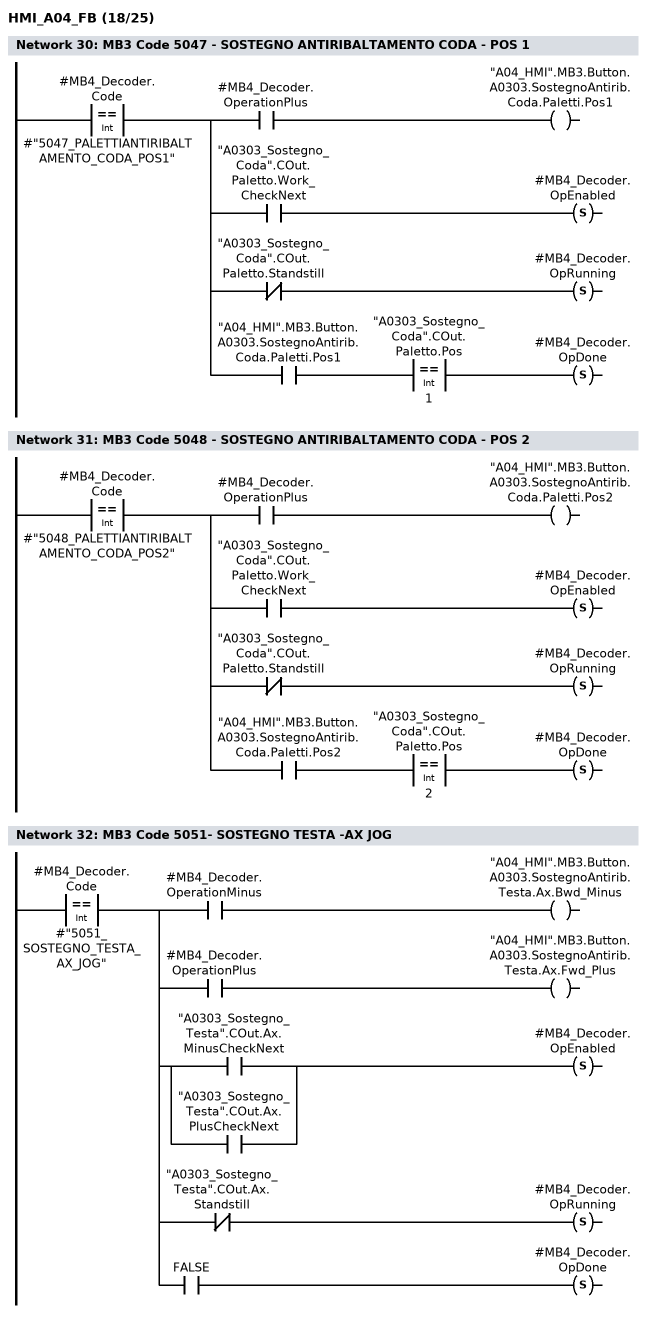
   RUNG wire#powerrail
      { S7_Templates := "SrcType := Int" } EQ_Contact(in1 := #MB4_Decoder.Code, in2 := #"5047_PALETTIANTIRIBALTAMENTO_CODA_POS1")
      wire#w1
      Contact( #MB4_Decoder.OperationPlus )
      Coil( "A04_HMI".MB3.Button.A0303.SostegnoAntirib.Coda.Paletti.Pos1 )
   END_RUNG
   RUNG wire#w1
      Contact( "A0303_Sostegno_Coda".COut.Paletto.Work_CheckNext )
      S_Coil( #MB4_Decoder.OpEnabled )
   END_RUNG
   RUNG wire#w1
      I_Contact( "A0303_Sostegno_Coda".COut.Paletto.Standstill )
      S_Coil( #MB4_Decoder.OpRunning )
   END_RUNG
   RUNG wire#w1
      Contact( "A04_HMI".MB3.Button.A0303.SostegnoAntirib.Coda.Paletti.Pos1 )
      { S7_Templates := "SrcType := Int" } EQ_Contact(in1 := "A0303_Sostegno_Coda".COut.Paletto.Pos, in2 := 1)
      S_Coil( #MB4_Decoder.OpDone )
   END_RUNG
   // the same network as SCL:
   #_w1 := #MB4_Decoder.Code = #"5047_PALETTIANTIRIBALTAMENTO_CODA_POS1";
   "A04_HMI".MB3.Button.A0303.SostegnoAntirib.Coda.Paletti.Pos1 := #_w1 AND #MB4_Decoder.OperationPlus;
   IF #_w1 AND "A0303_Sostegno_Coda".COut.Paletto.Work_CheckNext THEN #MB4_Decoder.OpEnabled := TRUE; END_IF;
   IF #_w1 AND NOT "A0303_Sostegno_Coda".COut.Paletto.Standstill THEN #MB4_Decoder.OpRunning := TRUE; END_IF;
   IF #_w1 AND "A04_HMI".MB3.Button.A0303.SostegnoAntirib.Coda.Paletti.Pos1 AND ("A0303_Sostegno_Coda".COut.Paletto.Pos = 1) THEN
       #MB4_Decoder.OpDone := TRUE;
   END_IF;
END_REGION

REGION Network 31: MB3 Code 5048 - SOSTEGNO ANTIRIBALTAMENTO CODA - POS 2
   RUNG wire#powerrail
      { S7_Templates := "SrcType := Int" } EQ_Contact(in1 := #MB4_Decoder.Code, in2 := #"5048_PALETTIANTIRIBALTAMENTO_CODA_POS2")
      wire#w1
      Contact( #MB4_Decoder.OperationPlus )
      Coil( "A04_HMI".MB3.Button.A0303.SostegnoAntirib.Coda.Paletti.Pos2 )
   END_RUNG
   RUNG wire#w1
      Contact( "A0303_Sostegno_Coda".COut.Paletto.Work_CheckNext )
      S_Coil( #MB4_Decoder.OpEnabled )
   END_RUNG
   RUNG wire#w1
      I_Contact( "A0303_Sostegno_Coda".COut.Paletto.Standstill )
      S_Coil( #MB4_Decoder.OpRunning )
   END_RUNG
   RUNG wire#w1
      Contact( "A04_HMI".MB3.Button.A0303.SostegnoAntirib.Coda.Paletti.Pos2 )
      { S7_Templates := "SrcType := Int" } EQ_Contact(in1 := "A0303_Sostegno_Coda".COut.Paletto.Pos, in2 := 2)
      S_Coil( #MB4_Decoder.OpDone )
   END_RUNG
   // the same network as SCL:
   #_w1 := #MB4_Decoder.Code = #"5048_PALETTIANTIRIBALTAMENTO_CODA_POS2";
   "A04_HMI".MB3.Button.A0303.SostegnoAntirib.Coda.Paletti.Pos2 := #_w1 AND #MB4_Decoder.OperationPlus;
   IF #_w1 AND "A0303_Sostegno_Coda".COut.Paletto.Work_CheckNext THEN #MB4_Decoder.OpEnabled := TRUE; END_IF;
   IF #_w1 AND NOT "A0303_Sostegno_Coda".COut.Paletto.Standstill THEN #MB4_Decoder.OpRunning := TRUE; END_IF;
   IF #_w1 AND "A04_HMI".MB3.Button.A0303.SostegnoAntirib.Coda.Paletti.Pos2 AND ("A0303_Sostegno_Coda".COut.Paletto.Pos = 2) THEN
       #MB4_Decoder.OpDone := TRUE;
   END_IF;
END_REGION

REGION Network 32: MB3 Code 5051- SOSTEGNO TESTA -AX JOG
   RUNG wire#powerrail
      { S7_Templates := "SrcType := Int" } EQ_Contact(in1 := #MB4_Decoder.Code, in2 := #"5051_SOSTEGNO_TESTA_AX_JOG")
      wire#w1
      Contact( #MB4_Decoder.OperationMinus )
      Coil( "A04_HMI".MB3.Button.A0303.SostegnoAntirib.Testa.Ax.Bwd_Minus )
   END_RUNG
   RUNG wire#w1
      Contact( #MB4_Decoder.OperationPlus )
      Coil( "A04_HMI".MB3.Button.A0303.SostegnoAntirib.Testa.Ax.Fwd_Plus )
   END_RUNG
   RUNG wire#w1
      Contact( "A0303_Sostegno_Testa".COut.Ax.MinusCheckNext )
      wire#w2
      S_Coil( #MB4_Decoder.OpEnabled )
   END_RUNG
   RUNG wire#w1
      Contact( "A0303_Sostegno_Testa".COut.Ax.PlusCheckNext )
   END_RUNG wire#w2
   RUNG wire#w1
      I_Contact( "A0303_Sostegno_Testa".COut.Ax.Standstill )
      S_Coil( #MB4_Decoder.OpRunning )
   END_RUNG
   RUNG wire#w1
      Contact( FALSE )
      S_Coil( #MB4_Decoder.OpDone )
   END_RUNG
   // the same network as SCL:
   #_w1 := #MB4_Decoder.Code = #"5051_SOSTEGNO_TESTA_AX_JOG";
   "A04_HMI".MB3.Button.A0303.SostegnoAntirib.Testa.Ax.Bwd_Minus := #_w1 AND #MB4_Decoder.OperationMinus;
   "A04_HMI".MB3.Button.A0303.SostegnoAntirib.Testa.Ax.Fwd_Plus := #_w1 AND #MB4_Decoder.OperationPlus;
   IF #_w1 AND ("A0303_Sostegno_Testa".COut.Ax.MinusCheckNext OR "A0303_Sostegno_Testa".COut.Ax.PlusCheckNext) THEN
       #MB4_Decoder.OpEnabled := TRUE;
   END_IF;
   IF #_w1 AND NOT "A0303_Sostegno_Testa".COut.Ax.Standstill THEN #MB4_Decoder.OpRunning := TRUE; END_IF;
   IF #_w1 AND FALSE THEN #MB4_Decoder.OpDone := TRUE; END_IF;
END_REGION

REGION Network 33: MB3 Code 5051- SOSTEGNO TESTA -AX - POS
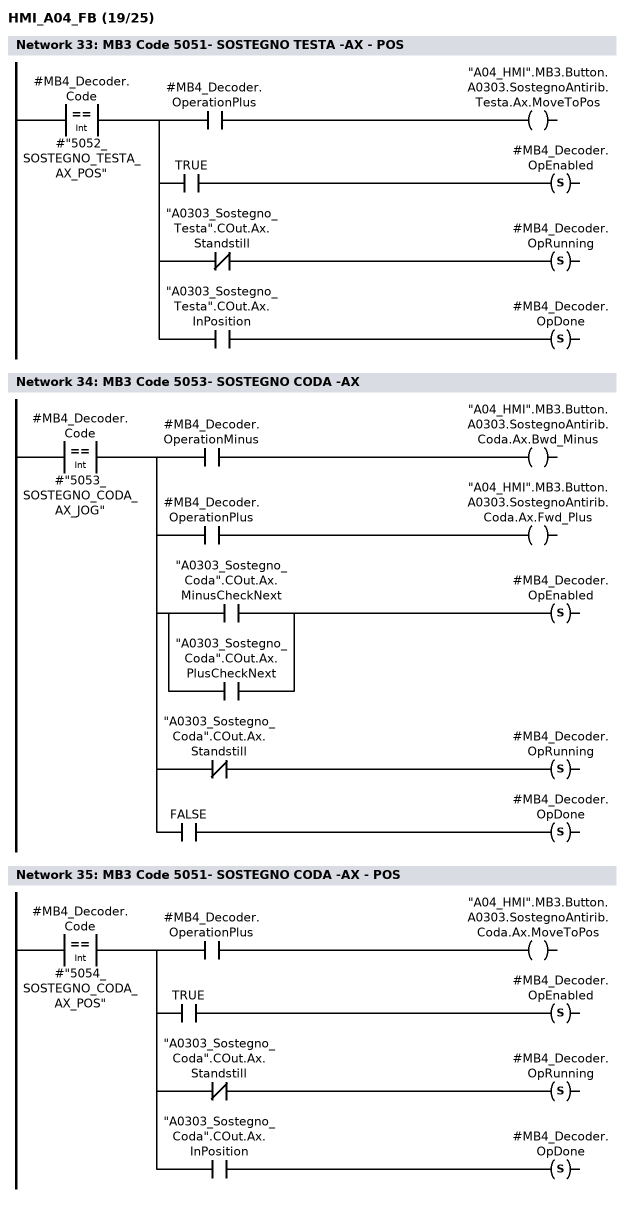
   RUNG wire#powerrail
      { S7_Templates := "SrcType := Int" } EQ_Contact(in1 := #MB4_Decoder.Code, in2 := #"5052_SOSTEGNO_TESTA_AX_POS")
      wire#w1
      Contact( #MB4_Decoder.OperationPlus )
      Coil( "A04_HMI".MB3.Button.A0303.SostegnoAntirib.Testa.Ax.MoveToPos )
   END_RUNG
   RUNG wire#w1
      Contact( TRUE )
      S_Coil( #MB4_Decoder.OpEnabled )
   END_RUNG
   RUNG wire#w1
      I_Contact( "A0303_Sostegno_Testa".COut.Ax.Standstill )
      S_Coil( #MB4_Decoder.OpRunning )
   END_RUNG
   RUNG wire#w1
      Contact( "A0303_Sostegno_Testa".COut.Ax.InPosition )
      S_Coil( #MB4_Decoder.OpDone )
   END_RUNG
   // the same network as SCL:
   #_w1 := #MB4_Decoder.Code = #"5052_SOSTEGNO_TESTA_AX_POS";
   "A04_HMI".MB3.Button.A0303.SostegnoAntirib.Testa.Ax.MoveToPos := #_w1 AND #MB4_Decoder.OperationPlus;
   IF #_w1 AND TRUE THEN #MB4_Decoder.OpEnabled := TRUE; END_IF;
   IF #_w1 AND NOT "A0303_Sostegno_Testa".COut.Ax.Standstill THEN #MB4_Decoder.OpRunning := TRUE; END_IF;
   IF #_w1 AND "A0303_Sostegno_Testa".COut.Ax.InPosition THEN #MB4_Decoder.OpDone := TRUE; END_IF;
END_REGION

REGION Network 34: MB3 Code 5053- SOSTEGNO CODA -AX
   RUNG wire#powerrail
      { S7_Templates := "SrcType := Int" } EQ_Contact(in1 := #MB4_Decoder.Code, in2 := #"5053_SOSTEGNO_CODA_AX_JOG")
      wire#w1
      Contact( #MB4_Decoder.OperationMinus )
      Coil( "A04_HMI".MB3.Button.A0303.SostegnoAntirib.Coda.Ax.Bwd_Minus )
   END_RUNG
   RUNG wire#w1
      Contact( #MB4_Decoder.OperationPlus )
      Coil( "A04_HMI".MB3.Button.A0303.SostegnoAntirib.Coda.Ax.Fwd_Plus )
   END_RUNG
   RUNG wire#w1
      Contact( "A0303_Sostegno_Coda".COut.Ax.MinusCheckNext )
      wire#w2
      S_Coil( #MB4_Decoder.OpEnabled )
   END_RUNG
   RUNG wire#w1
      Contact( "A0303_Sostegno_Coda".COut.Ax.PlusCheckNext )
   END_RUNG wire#w2
   RUNG wire#w1
      I_Contact( "A0303_Sostegno_Coda".COut.Ax.Standstill )
      S_Coil( #MB4_Decoder.OpRunning )
   END_RUNG
   RUNG wire#w1
      Contact( FALSE )
      S_Coil( #MB4_Decoder.OpDone )
   END_RUNG
   // the same network as SCL:
   #_w1 := #MB4_Decoder.Code = #"5053_SOSTEGNO_CODA_AX_JOG";
   "A04_HMI".MB3.Button.A0303.SostegnoAntirib.Coda.Ax.Bwd_Minus := #_w1 AND #MB4_Decoder.OperationMinus;
   "A04_HMI".MB3.Button.A0303.SostegnoAntirib.Coda.Ax.Fwd_Plus := #_w1 AND #MB4_Decoder.OperationPlus;
   IF #_w1 AND ("A0303_Sostegno_Coda".COut.Ax.MinusCheckNext OR "A0303_Sostegno_Coda".COut.Ax.PlusCheckNext) THEN
       #MB4_Decoder.OpEnabled := TRUE;
   END_IF;
   IF #_w1 AND NOT "A0303_Sostegno_Coda".COut.Ax.Standstill THEN #MB4_Decoder.OpRunning := TRUE; END_IF;
   IF #_w1 AND FALSE THEN #MB4_Decoder.OpDone := TRUE; END_IF;
END_REGION

REGION Network 35: MB3 Code 5051- SOSTEGNO CODA -AX - POS
   RUNG wire#powerrail
      { S7_Templates := "SrcType := Int" } EQ_Contact(in1 := #MB4_Decoder.Code, in2 := #"5054_SOSTEGNO_CODA_AX_POS")
      wire#w1
      Contact( #MB4_Decoder.OperationPlus )
      Coil( "A04_HMI".MB3.Button.A0303.SostegnoAntirib.Coda.Ax.MoveToPos )
   END_RUNG
   RUNG wire#w1
      Contact( TRUE )
      S_Coil( #MB4_Decoder.OpEnabled )
   END_RUNG
   RUNG wire#w1
      I_Contact( "A0303_Sostegno_Coda".COut.Ax.Standstill )
      S_Coil( #MB4_Decoder.OpRunning )
   END_RUNG
   RUNG wire#w1
      Contact( "A0303_Sostegno_Coda".COut.Ax.InPosition )
      S_Coil( #MB4_Decoder.OpDone )
   END_RUNG
   // the same network as SCL:
   #_w1 := #MB4_Decoder.Code = #"5054_SOSTEGNO_CODA_AX_POS";
   "A04_HMI".MB3.Button.A0303.SostegnoAntirib.Coda.Ax.MoveToPos := #_w1 AND #MB4_Decoder.OperationPlus;
   IF #_w1 AND TRUE THEN #MB4_Decoder.OpEnabled := TRUE; END_IF;
   IF #_w1 AND NOT "A0303_Sostegno_Coda".COut.Ax.Standstill THEN #MB4_Decoder.OpRunning := TRUE; END_IF;
   IF #_w1 AND "A0303_Sostegno_Coda".COut.Ax.InPosition THEN #MB4_Decoder.OpDone := TRUE; END_IF;
END_REGION

REGION Network 36: <<<<<<<<< A0304 STAZIONE 4>>>>>>>>>>>>>
END_REGION

REGION Network 37: MB3 Code 6001- NAVETTA - OP VAI A PRELIEVO
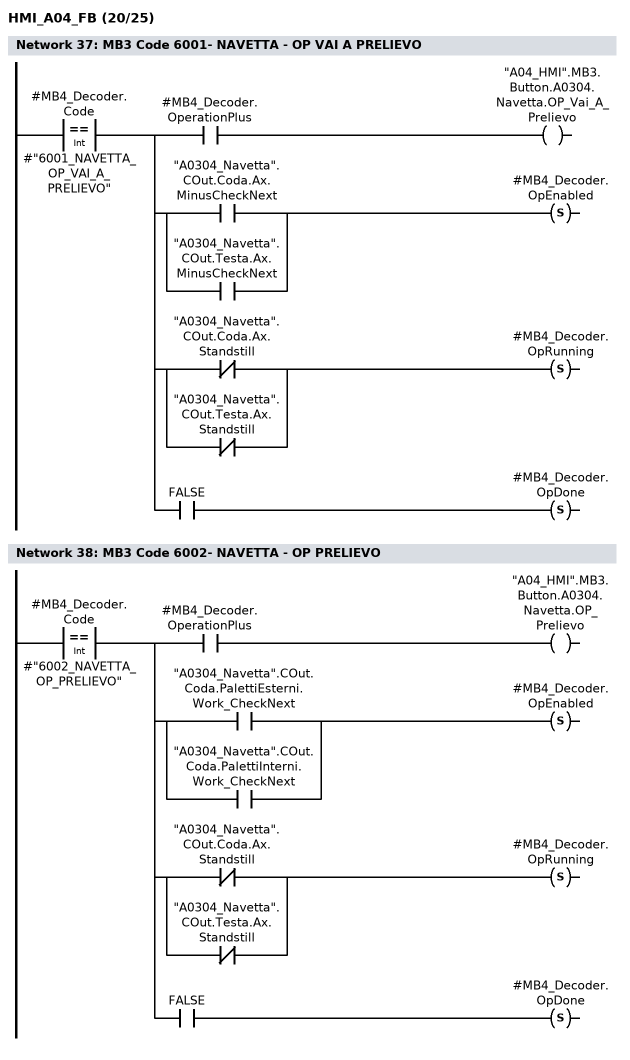
   RUNG wire#powerrail
      { S7_Templates := "SrcType := Int" } EQ_Contact(in1 := #MB4_Decoder.Code, in2 := #"6001_NAVETTA_OP_VAI_A_PRELIEVO")
      wire#w1
      Contact( #MB4_Decoder.OperationPlus )
      Coil( "A04_HMI".MB3.Button.A0304.Navetta.OP_Vai_A_Prelievo )
   END_RUNG
   RUNG wire#w1
      Contact( "A0304_Navetta".COut.Coda.Ax.MinusCheckNext )
      wire#w2
      S_Coil( #MB4_Decoder.OpEnabled )
   END_RUNG
   RUNG wire#w1
      Contact( "A0304_Navetta".COut.Testa.Ax.MinusCheckNext )
   END_RUNG wire#w2
   RUNG wire#w1
      I_Contact( "A0304_Navetta".COut.Coda.Ax.Standstill )
      wire#w3
      S_Coil( #MB4_Decoder.OpRunning )
   END_RUNG
   RUNG wire#w1
      I_Contact( "A0304_Navetta".COut.Testa.Ax.Standstill )
   END_RUNG wire#w3
   RUNG wire#w1
      Contact( FALSE )
      S_Coil( #MB4_Decoder.OpDone )
   END_RUNG
   // the same network as SCL:
   #_w1 := #MB4_Decoder.Code = #"6001_NAVETTA_OP_VAI_A_PRELIEVO";
   "A04_HMI".MB3.Button.A0304.Navetta.OP_Vai_A_Prelievo := #_w1 AND #MB4_Decoder.OperationPlus;
   IF #_w1 AND ("A0304_Navetta".COut.Coda.Ax.MinusCheckNext OR "A0304_Navetta".COut.Testa.Ax.MinusCheckNext) THEN
       #MB4_Decoder.OpEnabled := TRUE;
   END_IF;
   IF #_w1 AND (NOT "A0304_Navetta".COut.Coda.Ax.Standstill OR NOT "A0304_Navetta".COut.Testa.Ax.Standstill) THEN
       #MB4_Decoder.OpRunning := TRUE;
   END_IF;
   IF #_w1 AND FALSE THEN #MB4_Decoder.OpDone := TRUE; END_IF;
END_REGION

REGION Network 38: MB3 Code 6002- NAVETTA - OP PRELIEVO
   RUNG wire#powerrail
      { S7_Templates := "SrcType := Int" } EQ_Contact(in1 := #MB4_Decoder.Code, in2 := #"6002_NAVETTA_OP_PRELIEVO")
      wire#w1
      Contact( #MB4_Decoder.OperationPlus )
      Coil( "A04_HMI".MB3.Button.A0304.Navetta.OP_Prelievo )
   END_RUNG
   RUNG wire#w1
      Contact( "A0304_Navetta".COut.Coda.PalettiEsterni.Work_CheckNext )
      wire#w2
      S_Coil( #MB4_Decoder.OpEnabled )
   END_RUNG
   RUNG wire#w1
      Contact( "A0304_Navetta".COut.Coda.PalettiInterni.Work_CheckNext )
   END_RUNG wire#w2
   RUNG wire#w1
      I_Contact( "A0304_Navetta".COut.Coda.Ax.Standstill )
      wire#w3
      S_Coil( #MB4_Decoder.OpRunning )
   END_RUNG
   RUNG wire#w1
      I_Contact( "A0304_Navetta".COut.Testa.Ax.Standstill )
   END_RUNG wire#w3
   RUNG wire#w1
      Contact( FALSE )
      S_Coil( #MB4_Decoder.OpDone )
   END_RUNG
   // the same network as SCL:
   #_w1 := #MB4_Decoder.Code = #"6002_NAVETTA_OP_PRELIEVO";
   "A04_HMI".MB3.Button.A0304.Navetta.OP_Prelievo := #_w1 AND #MB4_Decoder.OperationPlus;
   IF #_w1 AND ("A0304_Navetta".COut.Coda.PalettiEsterni.Work_CheckNext OR "A0304_Navetta".COut.Coda.PalettiInterni.Work_CheckNext) THEN
       #MB4_Decoder.OpEnabled := TRUE;
   END_IF;
   IF #_w1 AND (NOT "A0304_Navetta".COut.Coda.Ax.Standstill OR NOT "A0304_Navetta".COut.Testa.Ax.Standstill) THEN
       #MB4_Decoder.OpRunning := TRUE;
   END_IF;
   IF #_w1 AND FALSE THEN #MB4_Decoder.OpDone := TRUE; END_IF;
END_REGION

REGION Network 39: MB3 Code 6003- NAVETTA - OP VAI A DEPOSITO
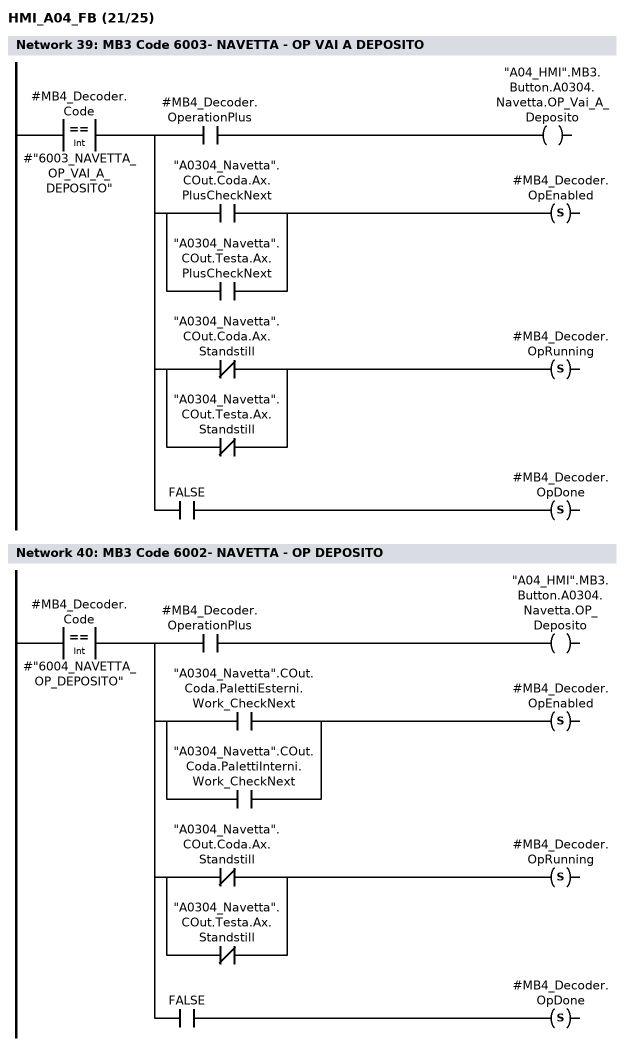
   RUNG wire#powerrail
      { S7_Templates := "SrcType := Int" } EQ_Contact(in1 := #MB4_Decoder.Code, in2 := #"6003_NAVETTA_OP_VAI_A_DEPOSITO")
      wire#w1
      Contact( #MB4_Decoder.OperationPlus )
      Coil( "A04_HMI".MB3.Button.A0304.Navetta.OP_Vai_A_Deposito )
   END_RUNG
   RUNG wire#w1
      Contact( "A0304_Navetta".COut.Coda.Ax.PlusCheckNext )
      wire#w2
      S_Coil( #MB4_Decoder.OpEnabled )
   END_RUNG
   RUNG wire#w1
      Contact( "A0304_Navetta".COut.Testa.Ax.PlusCheckNext )
   END_RUNG wire#w2
   RUNG wire#w1
      I_Contact( "A0304_Navetta".COut.Coda.Ax.Standstill )
      wire#w3
      S_Coil( #MB4_Decoder.OpRunning )
   END_RUNG
   RUNG wire#w1
      I_Contact( "A0304_Navetta".COut.Testa.Ax.Standstill )
   END_RUNG wire#w3
   RUNG wire#w1
      Contact( FALSE )
      S_Coil( #MB4_Decoder.OpDone )
   END_RUNG
   // the same network as SCL:
   #_w1 := #MB4_Decoder.Code = #"6003_NAVETTA_OP_VAI_A_DEPOSITO";
   "A04_HMI".MB3.Button.A0304.Navetta.OP_Vai_A_Deposito := #_w1 AND #MB4_Decoder.OperationPlus;
   IF #_w1 AND ("A0304_Navetta".COut.Coda.Ax.PlusCheckNext OR "A0304_Navetta".COut.Testa.Ax.PlusCheckNext) THEN
       #MB4_Decoder.OpEnabled := TRUE;
   END_IF;
   IF #_w1 AND (NOT "A0304_Navetta".COut.Coda.Ax.Standstill OR NOT "A0304_Navetta".COut.Testa.Ax.Standstill) THEN
       #MB4_Decoder.OpRunning := TRUE;
   END_IF;
   IF #_w1 AND FALSE THEN #MB4_Decoder.OpDone := TRUE; END_IF;
END_REGION

REGION Network 40: MB3 Code 6002- NAVETTA - OP DEPOSITO
   RUNG wire#powerrail
      { S7_Templates := "SrcType := Int" } EQ_Contact(in1 := #MB4_Decoder.Code, in2 := #"6004_NAVETTA_OP_DEPOSITO")
      wire#w1
      Contact( #MB4_Decoder.OperationPlus )
      Coil( "A04_HMI".MB3.Button.A0304.Navetta.OP_Deposito )
   END_RUNG
   RUNG wire#w1
      Contact( "A0304_Navetta".COut.Coda.PalettiEsterni.Work_CheckNext )
      wire#w2
      S_Coil( #MB4_Decoder.OpEnabled )
   END_RUNG
   RUNG wire#w1
      Contact( "A0304_Navetta".COut.Coda.PalettiInterni.Work_CheckNext )
   END_RUNG wire#w2
   RUNG wire#w1
      I_Contact( "A0304_Navetta".COut.Coda.Ax.Standstill )
      wire#w3
      S_Coil( #MB4_Decoder.OpRunning )
   END_RUNG
   RUNG wire#w1
      I_Contact( "A0304_Navetta".COut.Testa.Ax.Standstill )
   END_RUNG wire#w3
   RUNG wire#w1
      Contact( FALSE )
      S_Coil( #MB4_Decoder.OpDone )
   END_RUNG
   // the same network as SCL:
   #_w1 := #MB4_Decoder.Code = #"6004_NAVETTA_OP_DEPOSITO";
   "A04_HMI".MB3.Button.A0304.Navetta.OP_Deposito := #_w1 AND #MB4_Decoder.OperationPlus;
   IF #_w1 AND ("A0304_Navetta".COut.Coda.PalettiEsterni.Work_CheckNext OR "A0304_Navetta".COut.Coda.PalettiInterni.Work_CheckNext) THEN
       #MB4_Decoder.OpEnabled := TRUE;
   END_IF;
   IF #_w1 AND (NOT "A0304_Navetta".COut.Coda.Ax.Standstill OR NOT "A0304_Navetta".COut.Testa.Ax.Standstill) THEN
       #MB4_Decoder.OpRunning := TRUE;
   END_IF;
   IF #_w1 AND FALSE THEN #MB4_Decoder.OpDone := TRUE; END_IF;
END_REGION

REGION Network 41: MB3 Code 6004- NAVETTA -AX
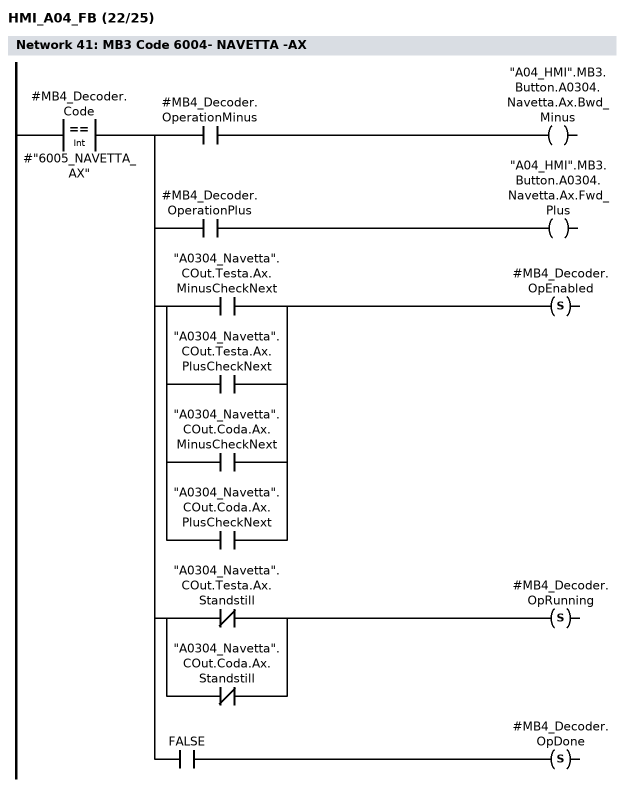
   RUNG wire#powerrail
      { S7_Templates := "SrcType := Int" } EQ_Contact(in1 := #MB4_Decoder.Code, in2 := #"6005_NAVETTA_AX")
      wire#w1
      Contact( #MB4_Decoder.OperationMinus )
      Coil( "A04_HMI".MB3.Button.A0304.Navetta.Ax.Bwd_Minus )
   END_RUNG
   RUNG wire#w1
      Contact( #MB4_Decoder.OperationPlus )
      Coil( "A04_HMI".MB3.Button.A0304.Navetta.Ax.Fwd_Plus )
   END_RUNG
   RUNG wire#w1
      Contact( "A0304_Navetta".COut.Testa.Ax.MinusCheckNext )
      wire#w2
      S_Coil( #MB4_Decoder.OpEnabled )
   END_RUNG
   RUNG wire#w1
      Contact( "A0304_Navetta".COut.Testa.Ax.PlusCheckNext )
   END_RUNG wire#w2
   RUNG wire#w1
      Contact( "A0304_Navetta".COut.Coda.Ax.MinusCheckNext )
   END_RUNG wire#w2
   RUNG wire#w1
      Contact( "A0304_Navetta".COut.Coda.Ax.PlusCheckNext )
   END_RUNG wire#w2
   RUNG wire#w1
      I_Contact( "A0304_Navetta".COut.Testa.Ax.Standstill )
      wire#w3
      S_Coil( #MB4_Decoder.OpRunning )
   END_RUNG
   RUNG wire#w1
      I_Contact( "A0304_Navetta".COut.Coda.Ax.Standstill )
   END_RUNG wire#w3
   RUNG wire#w1
      Contact( FALSE )
      S_Coil( #MB4_Decoder.OpDone )
   END_RUNG
   // the same network as SCL:
   #_w1 := #MB4_Decoder.Code = #"6005_NAVETTA_AX";
   "A04_HMI".MB3.Button.A0304.Navetta.Ax.Bwd_Minus := #_w1 AND #MB4_Decoder.OperationMinus;
   "A04_HMI".MB3.Button.A0304.Navetta.Ax.Fwd_Plus := #_w1 AND #MB4_Decoder.OperationPlus;
   IF #_w1 AND ("A0304_Navetta".COut.Testa.Ax.MinusCheckNext OR "A0304_Navetta".COut.Testa.Ax.PlusCheckNext OR "A0304_Navetta".COut.Coda.Ax.MinusCheckNext OR "A0304_Navetta".COut.Coda.Ax.PlusCheckNext) THEN
       #MB4_Decoder.OpEnabled := TRUE;
   END_IF;
   IF #_w1 AND (NOT "A0304_Navetta".COut.Testa.Ax.Standstill OR NOT "A0304_Navetta".COut.Coda.Ax.Standstill) THEN
       #MB4_Decoder.OpRunning := TRUE;
   END_IF;
   IF #_w1 AND FALSE THEN #MB4_Decoder.OpDone := TRUE; END_IF;
END_REGION

REGION Network 42: MB3 Code 6005 - NAVETTA - PALETTI INTERNI
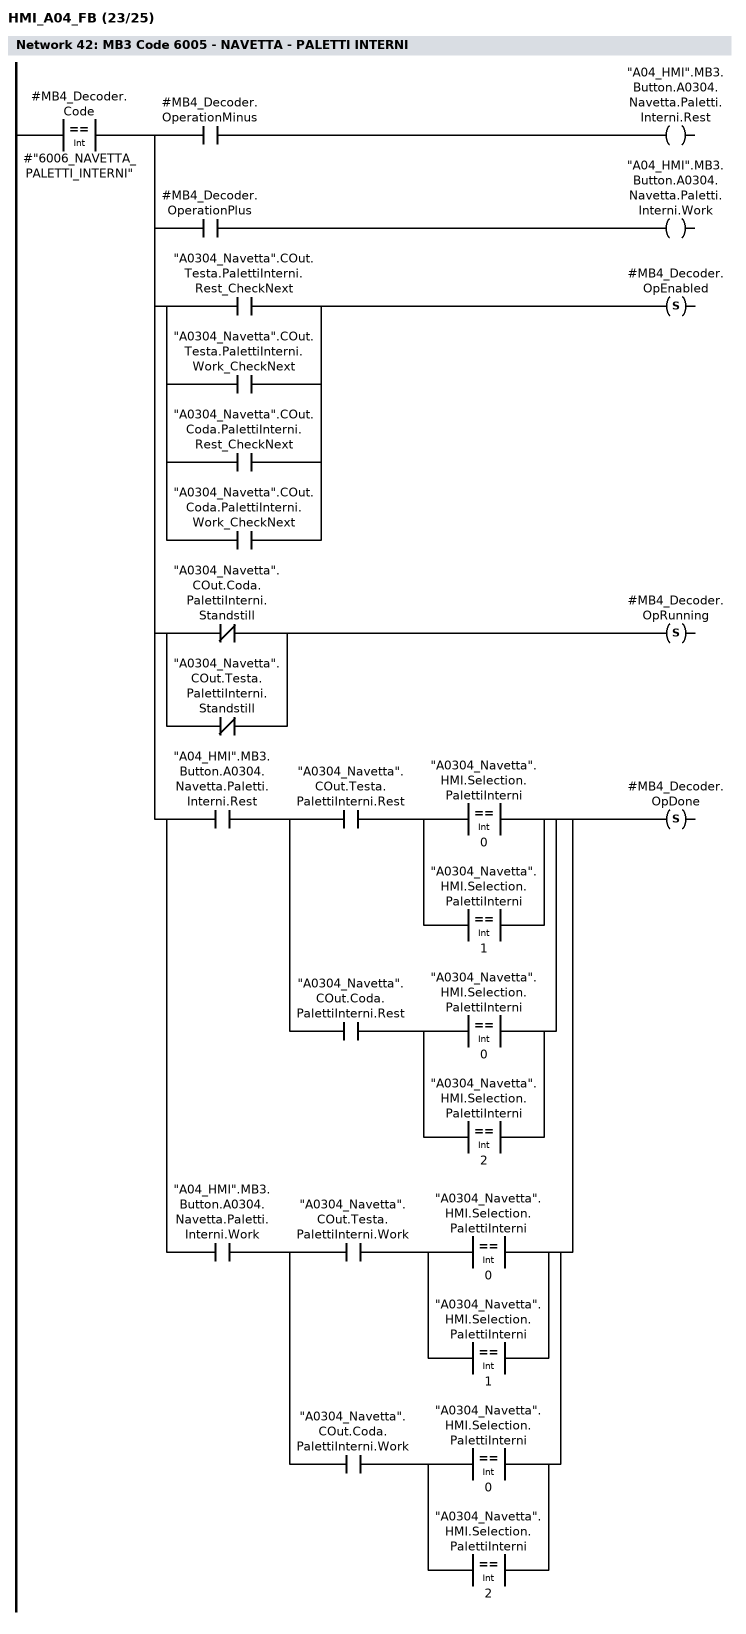
   RUNG wire#powerrail
      { S7_Templates := "SrcType := Int" } EQ_Contact(in1 := #MB4_Decoder.Code, in2 := #"6006_NAVETTA_PALETTI_INTERNI")
      wire#w1
      Contact( #MB4_Decoder.OperationMinus )
      Coil( "A04_HMI".MB3.Button.A0304.Navetta.Paletti.Interni.Rest )
   END_RUNG
   RUNG wire#w1
      Contact( #MB4_Decoder.OperationPlus )
      Coil( "A04_HMI".MB3.Button.A0304.Navetta.Paletti.Interni.Work )
   END_RUNG
   RUNG wire#w1
      Contact( "A0304_Navetta".COut.Testa.PalettiInterni.Rest_CheckNext )
      wire#w2
      S_Coil( #MB4_Decoder.OpEnabled )
   END_RUNG
   RUNG wire#w1
      Contact( "A0304_Navetta".COut.Testa.PalettiInterni.Work_CheckNext )
   END_RUNG wire#w2
   RUNG wire#w1
      Contact( "A0304_Navetta".COut.Coda.PalettiInterni.Rest_CheckNext )
   END_RUNG wire#w2
   RUNG wire#w1
      Contact( "A0304_Navetta".COut.Coda.PalettiInterni.Work_CheckNext )
   END_RUNG wire#w2
   RUNG wire#w1
      I_Contact( "A0304_Navetta".COut.Coda.PalettiInterni.Standstill )
      wire#w3
      S_Coil( #MB4_Decoder.OpRunning )
   END_RUNG
   RUNG wire#w1
      I_Contact( "A0304_Navetta".COut.Testa.PalettiInterni.Standstill )
   END_RUNG wire#w3
   RUNG wire#w1
      Contact( "A04_HMI".MB3.Button.A0304.Navetta.Paletti.Interni.Rest )
      wire#w4
      Contact( "A0304_Navetta".COut.Testa.PalettiInterni.Rest )
      wire#w5
      { S7_Templates := "SrcType := Int" } EQ_Contact(in1 := "A0304_Navetta".HMI.Selection.PalettiInterni, in2 := 0)
      wire#w6
      S_Coil( #MB4_Decoder.OpDone )
   END_RUNG
   RUNG wire#w5
      { S7_Templates := "SrcType := Int" } EQ_Contact(in1 := "A0304_Navetta".HMI.Selection.PalettiInterni, in2 := 1)
   END_RUNG wire#w6
   RUNG wire#w4
      Contact( "A0304_Navetta".COut.Coda.PalettiInterni.Rest )
      wire#w7
      { S7_Templates := "SrcType := Int" } EQ_Contact(in1 := "A0304_Navetta".HMI.Selection.PalettiInterni, in2 := 0)
   END_RUNG wire#w6
   RUNG wire#w7
      { S7_Templates := "SrcType := Int" } EQ_Contact(in1 := "A0304_Navetta".HMI.Selection.PalettiInterni, in2 := 2)
   END_RUNG wire#w6
   RUNG wire#w1
      Contact( "A04_HMI".MB3.Button.A0304.Navetta.Paletti.Interni.Work )
      wire#w8
      Contact( "A0304_Navetta".COut.Testa.PalettiInterni.Work )
      wire#w9
      { S7_Templates := "SrcType := Int" } EQ_Contact(in1 := "A0304_Navetta".HMI.Selection.PalettiInterni, in2 := 0)
   END_RUNG wire#w6
   RUNG wire#w9
      { S7_Templates := "SrcType := Int" } EQ_Contact(in1 := "A0304_Navetta".HMI.Selection.PalettiInterni, in2 := 1)
   END_RUNG wire#w6
   RUNG wire#w8
      Contact( "A0304_Navetta".COut.Coda.PalettiInterni.Work )
      wire#w10
      { S7_Templates := "SrcType := Int" } EQ_Contact(in1 := "A0304_Navetta".HMI.Selection.PalettiInterni, in2 := 0)
   END_RUNG wire#w6
   RUNG wire#w10
      { S7_Templates := "SrcType := Int" } EQ_Contact(in1 := "A0304_Navetta".HMI.Selection.PalettiInterni, in2 := 2)
   END_RUNG wire#w6
   // the same network as SCL:
   #_w1 := #MB4_Decoder.Code = #"6006_NAVETTA_PALETTI_INTERNI";
   "A04_HMI".MB3.Button.A0304.Navetta.Paletti.Interni.Rest := #_w1 AND #MB4_Decoder.OperationMinus;
   "A04_HMI".MB3.Button.A0304.Navetta.Paletti.Interni.Work := #_w1 AND #MB4_Decoder.OperationPlus;
   IF #_w1 AND ("A0304_Navetta".COut.Testa.PalettiInterni.Rest_CheckNext OR "A0304_Navetta".COut.Testa.PalettiInterni.Work_CheckNext OR "A0304_Navetta".COut.Coda.PalettiInterni.Rest_CheckNext OR "A0304_Navetta".COut.Coda.PalettiInterni.Work_CheckNext) THEN
       #MB4_Decoder.OpEnabled := TRUE;
   END_IF;
   IF #_w1 AND (NOT "A0304_Navetta".COut.Coda.PalettiInterni.Standstill OR NOT "A0304_Navetta".COut.Testa.PalettiInterni.Standstill) THEN
       #MB4_Decoder.OpRunning := TRUE;
   END_IF;
   IF #_w1 AND (("A04_HMI".MB3.Button.A0304.Navetta.Paletti.Interni.Rest AND (("A0304_Navetta".COut.Testa.PalettiInterni.Rest AND (("A0304_Navetta".HMI.Selection.PalettiInterni = 0) OR ("A0304_Navetta".HMI.Selection.PalettiInterni = 1))) OR ("A0304_Navetta".COut.Coda.PalettiInterni.Rest AND (("A0304_Navetta".HMI.Selection.PalettiInterni = 0) OR ("A0304_Navetta".HMI.Selection.PalettiInterni = 2))))) OR ("A04_HMI".MB3.Button.A0304.Navetta.Paletti.Interni.Work AND (("A0304_Navetta".COut.Testa.PalettiInterni.Work AND (("A0304_Navetta".HMI.Selection.PalettiInterni = 0) OR ("A0304_Navetta".HMI.Selection.PalettiInterni = 1))) OR ("A0304_Navetta".COut.Coda.PalettiInterni.Work AND (("A0304_Navetta".HMI.Selection.PalettiInterni = 0) OR ("A0304_Navetta".HMI.Selection.PalettiInterni = 2)))))) THEN
       #MB4_Decoder.OpDone := TRUE;
   END_IF;
END_REGION

REGION Network 43: MB3 Code 6006 - NAVETTA - PALETTI ESTERNI
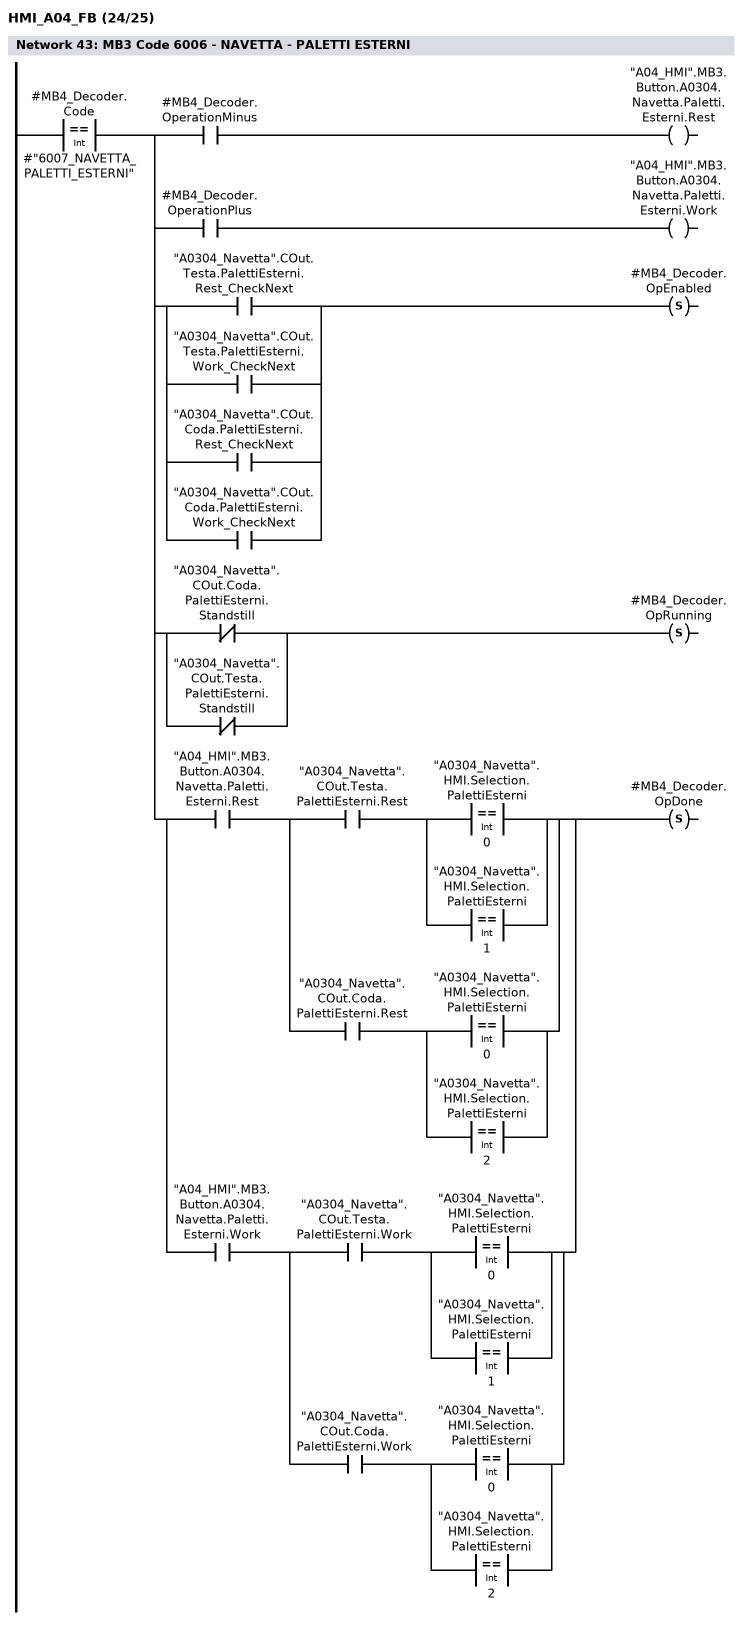
   RUNG wire#powerrail
      { S7_Templates := "SrcType := Int" } EQ_Contact(in1 := #MB4_Decoder.Code, in2 := #"6007_NAVETTA_PALETTI_ESTERNI")
      wire#w1
      Contact( #MB4_Decoder.OperationMinus )
      Coil( "A04_HMI".MB3.Button.A0304.Navetta.Paletti.Esterni.Rest )
   END_RUNG
   RUNG wire#w1
      Contact( #MB4_Decoder.OperationPlus )
      Coil( "A04_HMI".MB3.Button.A0304.Navetta.Paletti.Esterni.Work )
   END_RUNG
   RUNG wire#w1
      Contact( "A0304_Navetta".COut.Testa.PalettiEsterni.Rest_CheckNext )
      wire#w2
      S_Coil( #MB4_Decoder.OpEnabled )
   END_RUNG
   RUNG wire#w1
      Contact( "A0304_Navetta".COut.Testa.PalettiEsterni.Work_CheckNext )
   END_RUNG wire#w2
   RUNG wire#w1
      Contact( "A0304_Navetta".COut.Coda.PalettiEsterni.Rest_CheckNext )
   END_RUNG wire#w2
   RUNG wire#w1
      Contact( "A0304_Navetta".COut.Coda.PalettiEsterni.Work_CheckNext )
   END_RUNG wire#w2
   RUNG wire#w1
      I_Contact( "A0304_Navetta".COut.Coda.PalettiEsterni.Standstill )
      wire#w3
      S_Coil( #MB4_Decoder.OpRunning )
   END_RUNG
   RUNG wire#w1
      I_Contact( "A0304_Navetta".COut.Testa.PalettiEsterni.Standstill )
   END_RUNG wire#w3
   RUNG wire#w1
      Contact( "A04_HMI".MB3.Button.A0304.Navetta.Paletti.Esterni.Rest )
      wire#w4
      Contact( "A0304_Navetta".COut.Testa.PalettiEsterni.Rest )
      wire#w5
      { S7_Templates := "SrcType := Int" } EQ_Contact(in1 := "A0304_Navetta".HMI.Selection.PalettiEsterni, in2 := 0)
      wire#w6
      S_Coil( #MB4_Decoder.OpDone )
   END_RUNG
   RUNG wire#w5
      { S7_Templates := "SrcType := Int" } EQ_Contact(in1 := "A0304_Navetta".HMI.Selection.PalettiEsterni, in2 := 1)
   END_RUNG wire#w6
   RUNG wire#w4
      Contact( "A0304_Navetta".COut.Coda.PalettiEsterni.Rest )
      wire#w7
      { S7_Templates := "SrcType := Int" } EQ_Contact(in1 := "A0304_Navetta".HMI.Selection.PalettiEsterni, in2 := 0)
   END_RUNG wire#w6
   RUNG wire#w7
      { S7_Templates := "SrcType := Int" } EQ_Contact(in1 := "A0304_Navetta".HMI.Selection.PalettiEsterni, in2 := 2)
   END_RUNG wire#w6
   RUNG wire#w1
      Contact( "A04_HMI".MB3.Button.A0304.Navetta.Paletti.Esterni.Work )
      wire#w8
      Contact( "A0304_Navetta".COut.Testa.PalettiEsterni.Work )
      wire#w9
      { S7_Templates := "SrcType := Int" } EQ_Contact(in1 := "A0304_Navetta".HMI.Selection.PalettiEsterni, in2 := 0)
   END_RUNG wire#w6
   RUNG wire#w9
      { S7_Templates := "SrcType := Int" } EQ_Contact(in1 := "A0304_Navetta".HMI.Selection.PalettiEsterni, in2 := 1)
   END_RUNG wire#w6
   RUNG wire#w8
      Contact( "A0304_Navetta".COut.Coda.PalettiEsterni.Work )
      wire#w10
      { S7_Templates := "SrcType := Int" } EQ_Contact(in1 := "A0304_Navetta".HMI.Selection.PalettiEsterni, in2 := 0)
   END_RUNG wire#w6
   RUNG wire#w10
      { S7_Templates := "SrcType := Int" } EQ_Contact(in1 := "A0304_Navetta".HMI.Selection.PalettiEsterni, in2 := 2)
   END_RUNG wire#w6
   // the same network as SCL:
   #_w1 := #MB4_Decoder.Code = #"6007_NAVETTA_PALETTI_ESTERNI";
   "A04_HMI".MB3.Button.A0304.Navetta.Paletti.Esterni.Rest := #_w1 AND #MB4_Decoder.OperationMinus;
   "A04_HMI".MB3.Button.A0304.Navetta.Paletti.Esterni.Work := #_w1 AND #MB4_Decoder.OperationPlus;
   IF #_w1 AND ("A0304_Navetta".COut.Testa.PalettiEsterni.Rest_CheckNext OR "A0304_Navetta".COut.Testa.PalettiEsterni.Work_CheckNext OR "A0304_Navetta".COut.Coda.PalettiEsterni.Rest_CheckNext OR "A0304_Navetta".COut.Coda.PalettiEsterni.Work_CheckNext) THEN
       #MB4_Decoder.OpEnabled := TRUE;
   END_IF;
   IF #_w1 AND (NOT "A0304_Navetta".COut.Coda.PalettiEsterni.Standstill OR NOT "A0304_Navetta".COut.Testa.PalettiEsterni.Standstill) THEN
       #MB4_Decoder.OpRunning := TRUE;
   END_IF;
   IF #_w1 AND (("A04_HMI".MB3.Button.A0304.Navetta.Paletti.Esterni.Rest AND (("A0304_Navetta".COut.Testa.PalettiEsterni.Rest AND (("A0304_Navetta".HMI.Selection.PalettiEsterni = 0) OR ("A0304_Navetta".HMI.Selection.PalettiEsterni = 1))) OR ("A0304_Navetta".COut.Coda.PalettiEsterni.Rest AND (("A0304_Navetta".HMI.Selection.PalettiEsterni = 0) OR ("A0304_Navetta".HMI.Selection.PalettiEsterni = 2))))) OR ("A04_HMI".MB3.Button.A0304.Navetta.Paletti.Esterni.Work AND (("A0304_Navetta".COut.Testa.PalettiEsterni.Work AND (("A0304_Navetta".HMI.Selection.PalettiEsterni = 0) OR ("A0304_Navetta".HMI.Selection.PalettiEsterni = 1))) OR ("A0304_Navetta".COut.Coda.PalettiEsterni.Work AND (("A0304_Navetta".HMI.Selection.PalettiEsterni = 0) OR ("A0304_Navetta".HMI.Selection.PalettiEsterni = 2)))))) THEN
       #MB4_Decoder.OpDone := TRUE;
   END_IF;
END_REGION

REGION Network 44: MB3 Code6007- NAVETTA -AX - POS
